// SIMATIC STEP 7 (V5.x) project Combined_DEH_Config
// station: P_ADR_BUS
// station: Hardware
// station: SIMATIC 400(ATC-RSM)
// station: SIMATIC 400(OPC-OA)
// station: P_ADR_BUS
// station: Hardware
// program: S7 Program
// program: S7 Program(1)

SYMBOL_TABLE
"Constants_RSM"	DB 1	DB 1	// Sheet 2 (RSM)
"HISIGMTR-VALs"	DB 2	DB 2
"LOSIGMTR-VALs"	DB 3	DB 3
"AIN_VALs_VIB"	DB 4	FB 1	// DB for analog vibration inputs
"GAINBI-VALs"	DB 5	DB 5
"DELTAW-VALs"	DB 6	DB 6	// DELTAW contants
"HILOLMTV-VALs"	DB 7	DB 7
"HILOMTR-VALs"	DB 8	DB 8
"AVALGEN"	DB 9	DB 9	// Analog Value Generation
"DVALGEN"	DB 10	DB 10	// Digital Value Generation
"RUNAVG_VALs_369_370"	DB 11	FB 2	// RUNAVG_DB for blocks 369  and 370
"HISIGMTV-VALs"	DB 12	DB 12
"LOSIGMTV-VALs"	DB 13	DB 13
"XLIMIT_VALs"	DB 14	DB 14
"AIFCTGEN_Vals"	DB 15	DB 15
"MULTGB_VALs"	DB 16	DB 16
"SUM2W_VALs"	DB 17	DB 17
"RATEMTR_VALs"	DB 18	DB 18
"XSUM_VALs"	DB 19	DB 19
"XTRANSF_VALs"	DB 20	DB 20
"XHISEL_VALs"	DB 21	DB 21
"AIN_VALs_TEMP_100"	DB 22	FB 1
"DIVIDEGB_VALs"	DB 23	DB 23
"AIN_VALs_TEMP_286"	DB 24	FB 1
"POLY_VALs"	DB 25	DB 25
"SUM4W_VALs"	DB 26	DB 26
"SUM8W_VALs"	DB 27	DB 27
"AIN_VALs_TEMP_661"	DB 28	FB 1	// DB for analog temperature inputs
"AIN_VALs_PRESS_760"	DB 29	FB 1	// DB for pressure analog inputs
"RESETSUM_VALs"	DB 30	DB 30
"AIN_VALs_POS_25"	DB 31	FB 1
"XMULT_VALs"	DB 32	DB 32
"ATCTime_VALs"	DB 33	DB 33	// Time declaration for all the timers used
"DIGCNTNF_VALs"	DB 34	DB 34
"Constants_ATC"	DB 35	DB 35
"RUNAVG_VALs_235"	DB 36	FB 2
"AIN_VALs_POS_2"	DB 37	FB 1	// DB for analog position inputs
"RSMTime_VALs"	DB 38	DB 38
"TIMECHG_VALs"	DB 39	DB 39
"AIN"	FB 1	FB 1	// REAL conversion of analog input signals
"RUNAVG"	FB 2	FB 2	// Average of time based samples of input
"DRUMD16"	FB 3	FB 3	// Drum Controller with Sixteen Digital Outputs
"QC"	FC 1	FC 1	// QCHK1BAD
"Sheet 24 (ATC)"	FC 2	FC 2	// VIBRATION MONITOR
"TOD_Conversion"	FC 3	FC 3	// Supporting Block for Sheet 24 (ATC)
"Sheet 2 (RSM)"	FC 4	FC 4	// Initialization of constants in sheet 2 (RSM)
"TRANSF"	FC 5	FC 5	// Transfer between Two Analog Inputs
"AIFCTGEN"	FC 6	FC 6
"BIN_SEARCH"	FC 7	FC 7
"XHISEL"	FC 8	FC 8	// Selects the Greater of Two Gained and Biased Inputs
"QAVGN"	FC 10	FC 10	// Average up to Eight Analog Points
"HISIGMTR"	FC 11	FC 11	// High Signal Monitor with Reset Deadband and Fixed Limit
"LOSIGMTR"	FC 12	FC 12	// Low Signal Monitor with Reset Deadband and Fixed Limit
"GAINBI"	FC 14	FC 14	// Gain and Bias an Input
"DELTAW"	FC 15	FC 15	// Difference between Two Weighted Inputs
"HILOLMTV"	FC 16	FC 16	// High/Low Limiter, Variable Limits
"HILOMTR"	FC 18	FC 18	// High/Low Signal Monitor with Reset Deadband and Fixed Limits
"QTRANSN"	FC 19	FC 19	// Automatic transfer between analog inputs, select best quality
"DIVIDEGB"	FC 21	FC 21	// Divider with Gain and Bias
"POLY"	FC 22	FC 22	// Fifth Order Polynomial Equation
"QBLOCK"	FC 23	FC 23	// Output is equal to input and output quality is good.
"SUM8W"	FC 24	FC 24
"Sheet 3 (RSM)"	FC 25	FC 25	// FSST & TIMP & TSAT (Analog)
"Sheet 4 (RSM)"	FC 26	FC 26	// HP FILM & TICM & TMAX (Analog)
"Sheet 5 (RSM)"	FC 27	FC 27	// MWINC LOGIC (Digital)
"Sheet 7 (RSM)"	FC 28	FC 28	// HP INVALID LOGIC (Digital)
"RESETSUM"	FC 29	FC 29	// Summer with Reset
"Sheet 6 (RSM)"	FC 30	FC 30	// HP Stress Counters (Analog)
"HISIGMTV"	FC 31	FC 31	// High Signal Monitor, Reset Deadband and Variable Limits
"LOSIGMTV"	FC 32	FC 32	// Low Signal Monitor, Reset Deadband, Variable Limit
"HISEL10"	FC 33	FC 33	// High Signal Selector with 'TWO' Inputs
"XLIMIT"	FC 34	FC 34	// Limits a Gained and Biased Input
"LOSEL10"	FC 35	FC 35	// Low Signal Selector with 'TWO' Inputs
"Sheet 9 (RSM)"	FC 36	FC 36	// HP ROTSURF, T1-5 & TP1-4 (Analog)
"Sheet 8 (RSM)"	FC 37	FC 37	// HXFER & TWC (Analog)
"Sheet 10 (RSM)"	FC 38	FC 38	// HP TEMP T6-T15 (Analog)
"Sheet11 (RSM)"	FC 39	FC 39	// HP TEMP T16-T23 (Analog)
"MULTGB"	FC 40	FC 40	// Multiplier with Gain and Bias
"SUM2W"	FC 41	FC 41	// Sum of Two Weighted Inputs
"RATEMTR"	FC 42	FC 42	// Rate of Change Monitor, Reset Deadband, Fixed Rate Limit
"XSUM"	FC 43	FC 43	// Add Two Gained and Biased Inputs
"XTRANSF"	FC 44	FC 44	// Select a Gained and Biased Input Based on a Flag
"Sheet 12 (RSM)"	FC 45	FC 45	// HP TAVG (Analog)
"Sheet 13 (RSM)"	FC 46	FC 46	// HP EFFECTIVE TEMP DIFF. (Analog)
"Sheet 14 (RSM)"	FC 47	FC 47	// HP DRUM TIMERS (Analog)
"Sheet 15 (RSM)"	FC 48	FC 48	// HP TD1FT1-15 (Analog)
"Sheet 16 (RSM)"	FC 51	FC 51	// HP ANTIC. DIFF. (Analog)
"Sheet 17 (RSM)"	FC 53	FC 53	// % ROTOR STRESS LIMIT (Analog)
"XMULT"	FC 54	FC 54	// Multiples Two Gained and Biased Inputs
"Sheet 18 (RSM)"	FC 55	FC 55	// SMW INC/DEC (Analog)
"Sheet 19 (RSM)"	FC 57	FC 57	// TBP (Analog)
"Sheet 20 (RSM)"	FC 58	FC 58	// MWINCR (Analog)
"Sheet 21 (RSM)"	FC 59	FC 59	// ATC RATE & LOAD RESERVE (Analog)
"SUM4W"	FC 60	FC 60
"Sheet 22 (RSM)"	FC 61	FC 61	// REQ. STM CHEST METAL TEMP (Analog)
"Sheet 23 (RSM)"	FC 62	FC 62	// HP ROTOR STRESS LIMIT (Digital)
"Sheet 24 (RSM)"	FC 63	FC 63	// ATC TARGET (Analog)
"Sheet 25 (RSM)"	FC 64	FC 64	// TRANSFER DELAY (Digital)
"Sheet 26 (RSM)"	FC 65	FC 65	// LADDERS 35, 128, RESONANCE RANGE LOGIC (Digital)
"Sheet 28 (RSM)"	FC 66	FC 66	// LADDERS 22, 500, 600, DIGITAL POINTERS TMAX & TWC LOGIC (Digital)
"Sheet 29 (RSM)"	FC 67	FC 67	// LADDERS 29, 31, 500, FIRST STAGE STM > 75 *C (Digital)
"Sheet 27 (RSM)"	FC 68	FC 68	// LADDERS 43, 129, RTSHOLD (Digital)
"Sheet 30 (RSM)"	FC 69	FC 69	// LADDER 126, SYNC LOGIC & OVERRIDE (Digital)
"Sheet 31 (RSM)"	FC 70	FC 70	// LADDER 33, ANTIC HP STRESS > LIMIT (Digital)
"Sheet 32 (RSM)"	FC 71	FC 71	// LADDERS 37, 125, 130, SYNC LOGIC & OVERRIDE (Digital)
"Sheet 33 (RSM)"	FC 72	FC 72	// LADDER 124, 127, SYNC LOGIC & TVGVINIT (Digital)
"Sheet 34 (RSM)"	FC 73	FC 73	// LADDERS 122, 123, 135, SET SPEED PLATEAU (Digital)
"Sheet 35 (RSM)"	FC 74	FC 74	// LADDER 120, 121, P15 ALARMS ESTIMATE ROLL TIME LOGIC & ATC VPL (Digital)
"Sheet 36 (RSM)"	FC 75	FC 75	// LADDER 41, 119, P15 ALARMS (Digital)
"Sheet 37 (RSM)"	FC 76	FC 76	// GENERATOR AND EXCITOR TEMPERATURES (Analog)
"Sheet 2 (ATC)"	FC 77	FC 77	// LADDER 500, SENSOR FAIL (Digital)
"Sheet 3 (ATC)"	FC 78	FC 78	// SENSOR FAIL (Digital)
"DIGCNTNF"	FC 79	FC 79	// Digital Counter with Flag
"Sheet 4 (ATC)"	FC 81	FC 81	// LADDERS 1, 3 (Digital)
"Sheet 5 (ATC)"	FC 82	FC 82	// LADDERS 3, 5, 9, 600, P00M01-M11 (Digital)
"Sheet 6 (ATC)"	FC 83	FC 83	// LADDERS 7, 9, 13, ATC PERMISSIVE (Digital)
"Sheet 7 (ATC)"	FC 84	FC 84	// LADDER 81. LOOPS 27, 33. WATER COOLED GENERATOR (Analog)
"Sheet 8 (ATC)"	FC 85	FC 85	// LADDERS 91, 108, 133, GENERATOR ANNUNCIATOR (Digital)
"Sheet 9 (ATC)"	FC 86	FC 86	// LADDERS 81,83,85,87,109,130. LOOPS 28-30. EXMON & COOLGSHI & P09MXX  (Digital)
"Sheet 10 (ATC)"	FC 87	FC 87	// LADDERS 31, 34, 36, GENERATOR CALCULATIONS (Analog)
"Sheet 11 (ATC)"	FC 88	FC 88	// LADDERS 15, 17, 18. LOOPS 2, 3. STEAM CHEST - OIL COOLER MONITOR (Analog)
"2xHISIGMTV, QC"	FC 89	FC 89	// Supporting block for sheet 12, 24 (ATC)
"Sheet 12 (ATC)"	FC 91	FC 91	// BEARING METAL TEMPERATURES (Analog)
"Sheet 13 (ATC)"	FC 92	FC 92	// BEARING METAL, OIL COOLER - P08MXX (Digital)
"Sheet 14 (ATC)"	FC 93	FC 93	// BEARING METAL - P08M05, 8 (Digital)
"Sheet 15 (ATC)"	FC 94	FC 94	// ROTOR POSITION, DIFF EXPANSION (Analog)
"Sheet 16 (ATC)"	FC 95	FC 95	// ROTOR POSITION DIFFERENTIAL EXPANSION P11MXX (Digital)
"Sheet 17 (ATC)"	FC 96	FC 96	// LOOPS 39, 40, 41. CONDENSOR PRESS LP EXH HOOD (Analog)
"Sheet 18 (ATC)"	FC 97	FC 97	// LADDERS 89, 90, 189, 190. GLAND, EXH, VAC - P10MXX (Digital)
"Sheet 19 (ATC)"	FC 98	FC 98	// BRG TEMPERATURE HIGH & VBINC (Digital)
"Sheet 20 (ATC)"	FC 99	FC 99	// VIBRATION LIMIT (Analog)
"Sheet 21 (ATC)"	FC 100	FC 100	// LADDERS 302,304,306,400. VIBRATION ALARM AND TRIP (Digital)
"Sheet 22 (ATC)"	FC 101	FC 101	// LADDERS 32, 33, 41. VIBRATION RUNUP / RUNDOWN LOGIC (Digital)
"Sheet 23 (ATC)"	FC 102	FC 102	// LADDER 39. VIBRATION RUNDOWN / RUNBACK LOGIC (Digital)
"3xHISIGMTV, 1xLOSIGMTV"	FC 103	FC 103
"3xLOSIGMTV, 1xHISIGMTV"	FC 104	FC 104
"SCALE"	FC 105	FC 105	// Scaling Values
"Sheet 25 (ATC)"	FC 106	FC 106	// SPEED RESONANT RANGE MONITOR (Analog)
"Sheet 26 (ATC)"	FC 107	FC 107	// LADDERS 150, 420. VIBRATION SPEED REF LOGIC (Digital)
"Sheet 27 (ATC)"	FC 108	FC 108	// VIBRATION RUNBACK SPEED REF (Analog)
"Sheet 28 (ATC)"	FC 109	FC 109	// LADDERS 30, 43, 307, 308, 309. VIBRATION RUNUP/RUNTHRU LOGIC (Digital)
"Sheet 29 (ATC)"	FC 110	FC 110	// VIBRATION RUN THRU REF (Analog)
"Sheet 30 (ATC)"	FC 111	FC 111	// VIBRATION SPEED REF (Analog)
"Sheet 31 (ATC)"	FC 112	FC 112	// LOOPS 18, 19. WATER DETECTION (Analog)
"Sheet 32 (ATC)"	FC 113	FC 113	// LADDERS 49, 51, 53. DRAIN VALVE LOGIC (Digital)
"DT_TOD"	FC 115	FC 115	// DT to TOD
"SUBB24"	FC 116	FC 116	// Supporting block for sheet 24 (ATC)
"TIMECHG"	FC 117	FC 117	// Check Real-Time Clock, Set Flags
"Sheet 33 (ATC)"	FC 118	FC 118	// LOOPS 4, 5 (Analog)
"Sheet 34 (ATC)"	FC 119	FC 119	// LADDERS 19, 21, 23, 25, 27. TURNING GEAR - P03MXX (Digital)
"Sheet 35 (ATC)"	FC 120	FC 120	// LOOPS 6, 60. THRUST BEARING, ROTOR ECCEN. (Analog)
"Sheet 36 (ATC)"	FC 121	FC 121	// LADDERS 27, 600. ATC PLATEAU FLAGS (Digital)
"Sheet 37 (ATC)"	FC 122	FC 122	// OVERRIDE LOGIC (Analog)
"Sheet 38 (ATC)"	FC 123	FC 123	// OVERRIDE LOGIC (Digital)
"Sheet 39 (ATC)"	FC 124	FC 124	// OVERRIDE LOGIC (Digital)
"Sheet 40 (ATC)"	FC 125	FC 125	// LADDERS 200, 201, 203, 220. REQUEST TRIP P07MXX (Digital)
"Sheet 41 (ATC)"	FC 126	FC 126	// LADDERS 201, 202, 203. HOLD 1 & 2 - P07M13 (Digital)
"Sheet 42 (ATC)"	FC 127	FC 127	// LADDERS 110, 111, 112, 113. OVERRIDE & P07M12 (Digital)
"Sheet 43 (ATC)"	FC 128	FC 128	// LADDERS 11, 113, 114. HOLD LOAD & P07M09 - 14 (Digital)
"Sheet 44 (ATC)"	FC 129	FC 129	// LADDERS 115, 116. HOLD WS & P07M02 - 04 (Digital)
"Sheet 45 (ATC)"	FC 130	FC 130	// LADDERS 117, 118. LOAD RATE INC/DEC P07M05 - 08 (Digital)
"Sheet 47 (ATC)"	FC 131	FC 131	// LADDERS 118, 192. P00M00A-G (Digital)
"Sheet 46 (ATC)"	FC 132	FC 132	// LOOPS 63, 65. LOAD RATE (Analog)
"Sheet 48_49 (ATC)"	FC 133	FC 133	// Initialization of ATC constants from AVALGEN DB
"ASSAP"	I 0.0	BOOL	//  (ATC) - (FieldIO4-M1)
"BOPL"	I 0.1	BOOL	//  (ATC) - (FieldIO4-M1)
"BVAP"	I 0.2	BOOL	//  (ATC) - (FieldIO4-M1)
"DVSAP"	I 0.3	BOOL	//  (ATC) - (FieldIO4-M1)
"EHFPL"	I 0.4	BOOL	//  (ATC) - (FieldIO4-M1)
"EHSO"	I 0.5	BOOL	//  (ATC) - (FieldIO4-M1)
"GDOGF"	I 0.6	BOOL	//  (ATC) - (FieldIO4-M1)
"GVRNLV"	I 0.7	BOOL	//  (ATC) - (FieldIO4-M1)
"HPDVC"	I 1.0	BOOL	//  (ATC) - (FieldIO4-M1)
"HPDVO"	I 1.1	BOOL	//  (ATC) - (FieldIO4-M1)
"MBCSU"	I 1.2	BOOL	//  (ATC) - (FieldIO4-M1)
"MELIT"	I 1.3	BOOL	//  (ATC) - (FieldIO4-M1)
"MVHPIT"	I 1.4	BOOL	//  (ATC) - (FieldIO4-M1)
"OEPIT"	I 1.5	BOOL	//  (ATC) - (FieldIO4-M1)
"RSBC"	I 1.6	BOOL	//  (ATC) - (FieldIO4-M1)
"RSBSU"	I 1.7	BOOL	//  (ATC) - (FieldIO4-M1)
"TGE"	I 2.0	BOOL	//  (ATC) - (FieldIO5-M1)
"VRO"	I 2.1	BOOL	//  (ATC) - (FieldIO5-M1)
"VROUS"	I 2.2	BOOL	//  (ATC) - (FieldIO5-M1)
"VRSOTP"	I 2.3	BOOL	//  (ATC) - (FieldIO5-M1)
"CAB4T1_W"	IW 512	WORD	//  (RSM) - (FieldIO4-M3)
"CNDP1_W"	IW 514	WORD	//  (RSM) - (FieldIO4-M3)
"FSST1_W"	IW 516	WORD	//  (RSM) - (FieldIO4-M3)
"B1T1_W"	IW 518	WORD	//  (ATC) - (FieldIO4-M3)
"B2T1_W"	IW 520	WORD	//  (ATC) - (FieldIO4-M3)
"B3T1_W"	IW 522	WORD	//  (ATC) - (FieldIO4-M3)
"B4T1_W"	IW 524	WORD	//  (ATC) - (FieldIO4-M3)
"B5T1_W"	IW 526	WORD	//  (ATC) - (FieldIO4-M3)
"B6T1_W"	IW 528	WORD	//  (ATC) - (FieldIO4-M4)
"RP1_W"	IW 530	WORD	//  (ATC) - (FieldIO4-M4)
"TBFCT1_W"	IW 532	WORD	//  (ATC) - (FieldIO4-M4)
"TBFLT1_W"	IW 534	WORD	//  (ATC) - (FieldIO4-M4)
"TBRCT1_W"	IW 536	WORD	//  (ATC) - (FieldIO4-M4)
"TBRLT1_W"	IW 538	WORD	//  (ATC) - (FieldIO4-M4)
"VB9_W"	IW 540	WORD	//  (ATC) - (FieldIO4-M4)
"FSMT1_W"	IW 542	WORD	//  (RSM) - (FieldIO4-M4)
"B7T_W"	IW 544	WORD	//  (ATC) - (FieldIO4-M5)
"B8T_W"	IW 546	WORD	//  (ATC) - (FieldIO4-M5)
"B9T_W"	IW 548	WORD	//  (ATC) - (FieldIO4-M5)
"B10T_W"	IW 550	WORD	//  (ATC) - (FieldIO4-M5)
"CAB5T1_W"	IW 552	WORD	//  (ATC) - (FieldIO4-M5)
"CAB5T2_W"	IW 554	WORD	//  (ATC) - (FieldIO4-M5)
"CASEXP_W"	IW 556	WORD	//  (ATC) - (FieldIO4-M5)
"DEGEN_W"	IW 558	WORD	//  (ATC) - (FieldIO4-M5)
"VB1_W"	IW 560	WORD	//  (ATC) - (FieldIO4-M6)
"VB2_W"	IW 562	WORD	//  (ATC) - (FieldIO4-M6)
"VB3_W"	IW 564	WORD	//  (ATC) - (FieldIO4-M6)
"VB4_W"	IW 566	WORD	//  (ATC) - (FieldIO4-M6)
"VB5_W"	IW 568	WORD	//  (ATC) - (FieldIO4-M6)
"VB6_W"	IW 570	WORD	//  (ATC) - (FieldIO4-M6)
"VB7_W"	IW 572	WORD	//  (ATC) - (FieldIO4-M6)
"VB8_W"	IW 574	WORD	//  (ATC) - (FieldIO4-M6)
"CAB4T2_W"	IW 576	WORD	//  (RSM) - (FieldIO5-M3)
"CNDP2_W"	IW 578	WORD	//  (RSM) - (FieldIO5-M3)
"FSST2_W"	IW 580	WORD	//  (RSM) - (FieldIO5-M3)
"B1T2_W"	IW 582	WORD	//  (ATC) - (FieldIO5-M3)
"B2T2_W"	IW 584	WORD	//  (ATC) - (FieldIO5-M3)
"B3T2_W"	IW 586	WORD	//  (ATC) - (FieldIO5-M3)
"B4T2_W"	IW 588	WORD	//  (ATC) - (FieldIO5-M3)
"B5T2_W"	IW 590	WORD	//  (ATC) - (FieldIO5-M3)
"B6T2_W"	IW 592	WORD	//  (ATC) - (FieldIO5-M4)
"RP2_W"	IW 594	WORD	//  (ATC) - (FieldIO5-M4)
"TBFCT2_W"	IW 596	WORD	//  (ATC) - (FieldIO5-M4)
"TBFLT2_W"	IW 598	WORD	//  (ATC) - (FieldIO5-M4)
"TBRCT2_W"	IW 600	WORD	//  (ATC) - (FieldIO5-M4)
"TBRLT2_W"	IW 602	WORD	//  (ATC) - (FieldIO5-M4)
"VB10_W"	IW 604	WORD	//  (ATC) - (FieldIO5-M4)
"LPGST_W"	IW 606	WORD	//  (RSM) - (FieldIO5-M4)
"EHFLT_W"	IW 608	WORD	//  (ATC) - (FieldIO5-M5)
"HPBMIDT_W"	IW 610	WORD	//  (ATC) - (FieldIO5-M5)
"HPCMIDT_W"	IW 612	WORD	//  (ATC) - (FieldIO5-M5)
"LP1GNT_W"	IW 614	WORD	//  (ATC) - (FieldIO5-M5)
"LP1GVT_W"	IW 616	WORD	//  (ATC) - (FieldIO5-M5)
"LP2GNT_W"	IW 618	WORD	//  (ATC) - (FieldIO5-M5)
"LP2GVT_W"	IW 620	WORD	//  (ATC) - (FieldIO5-M5)
"ROTECC_W"	IW 622	WORD	//  (ATC) - (FieldIO5-M5)
"OCIT_W"	IW 624	WORD	//  (RSM) - (FieldIO5-M6)
"OCOT_W"	IW 626	WORD	//  (RSM) - (FieldIO5-M6)
"TIMPRAT"	M 0.1	BOOL	// Sheet 3 (RSM)
"Z061"	M 0.2	BOOL	// Sheet 3 (RSM)
"Z060"	M 0.3	BOOL	// Sheet 3 (RSM)
"Z115"	M 0.4	BOOL	// Sheet 28 (RSM)
"SELC06"	M 0.5	BOOL	// Sheet 28 (RSM)
"X66D"	M 0.6	BOOL	// Sheet 4 (RSM)
"X67D"	M 0.7	BOOL	// Sheet 4 (RSM)
"X08A"	M 1.0	BOOL	// Sheet 4 (RSM)
"Z121"	M 1.1	BOOL	// Sheet 4 (RSM)
"Z133"	M 1.2	BOOL	// Sheet 4 (RSM)
"Z745"	M 1.3	BOOL	// Sheet 5 (RSM)
"Z747"	M 1.4	BOOL	// Sheet 5 (RSM)
"X08F"	M 1.5	BOOL	// Sheet 5 (RSM)
"X08E"	M 1.6	BOOL	// Sheet 5 (RSM)
"Z135"	M 1.7	BOOL	// Sheet 5 (RSM)
"Z393"	M 2.0	BOOL	// Sheet 19 (RSM)
"Z395"	M 2.1	BOOL	// Sheet 19 (RSM)
"Z398"	M 2.2	BOOL	// Sheet 19 (RSM)
"Z600"	M 2.3	BOOL	// Sheet 21 (RSM)
"BR"	M 2.4	BOOL	// Sheet 12 (OPC)
"Z599"	M 2.5	BOOL	// Sheet 21 (RSM)
"BR4"	M 2.6	BOOL	// Sheet 28 (RSM)
"F5MNLCTL"	M 2.7	BOOL	// Sheet 8 (RSM)
"Z272"	M 3.0	BOOL	// Sheet 6 (RSM)
"Z274"	M 3.1	BOOL	// Sheet 6 (RSM)
"WSFAIL"	M 3.2	BOOL	// Sheet 5 (OPC)
"HPINV"	M 3.3	BOOL	// Sheet 6 (RSM)
"RTRSWSFL"	M 3.4	BOOL	// Sheet 6 (RSM)
"Z268"	M 3.5	BOOL	// Sheet 7 (RSM)
"Z269"	M 3.6	BOOL	// Sheet 7 (RSM)
"Z123"	M 3.7	BOOL	// Sheet 7 (RSM)
"Z124"	M 4.0	BOOL	// Sheet 7 (RSM)
"P01M05"	M 4.1	BOOL	// Sheet 7 (RSM)
"Z131"	M 4.2	BOOL	// Sheet 7 (RSM)
"RESTART"	M 4.3	BOOL	// Sheet 7 (RSM)
"TIMPFAIL"	M 4.4	BOOL	// Sheet 7 (RSM)
"BRN4"	M 4.5	BOOL	// Sheet 28 (RSM)
"OUT_180"	M 4.6	BOOL	// Sheet 7 (RSM)
"X08D"	M 4.7	BOOL	// Sheet 6 (RSM)
"OUT_270"	M 5.0	BOOL	// Sheet 6 (RSM)
"T5SEC"	M 5.1	BOOL	// Sheet 6 (RSM)
"XFER"	M 5.2	BOOL	// Sheet 28 (RSM)
"OUT_221"	M 5.3	BOOL	// Sheet 8 (RSM)
"Z228"	M 5.4	BOOL	// Sheet 8 (RSM)
"X10G"	M 5.5	BOOL	// Sheet 11 (RSM)
"A275"	M 5.7	BOOL	// Sheet 14 (RSM)
"B275"	M 6.0	BOOL	// Sheet 14 (RSM)
"C275"	M 6.1	BOOL	// Sheet 14 (RSM)
"D275"	M 6.2	BOOL	// Sheet 14 (RSM)
"E275"	M 6.3	BOOL	// Sheet 14 (RSM)
"F275"	M 6.4	BOOL	// Sheet 14 (RSM)
"G275"	M 6.5	BOOL	// Sheet 14 (RSM)
"H275"	M 6.6	BOOL	// Sheet 14 (RSM)
"I275"	M 6.7	BOOL	// Sheet 14 (RSM)
"J275"	M 7.0	BOOL	// Sheet 14 (RSM)
"K275"	M 7.1	BOOL	// Sheet 14 (RSM)
"L275"	M 7.2	BOOL	// Sheet 14 (RSM)
"M275"	M 7.3	BOOL	// Sheet 14 (RSM)
"N275"	M 7.4	BOOL	// Sheet 14 (RSM)
"O275"	M 7.5	BOOL	// Sheet 14 (RSM)
"X11L"	M 7.6	BOOL	// Sheet 17 (RSM)
"X73K"	M 7.7	BOOL	// Sheet 17 (RSM)
"X11P"	M 8.0	BOOL	// Sheet 17 (RSM)
"X11T"	M 8.1	BOOL	// Sheet 17 (RSM)
"X11N"	M 8.2	BOOL	// Sheet 17 (RSM)
"X11R"	M 8.3	BOOL	// Sheet 17 (RSM)
"X11V"	M 8.4	BOOL	// Sheet 17 (RSM)
"X09L"	M 8.5	BOOL	// Sheet 17 (RSM)
"X09K"	M 8.6	BOOL	// Sheet 17 (RSM)
"X67A"	M 8.7	BOOL	// Sheet 17 (RSM)
"X14M"	M 9.0	BOOL	// Sheet 18 (RSM)
"X14Q"	M 9.1	BOOL	// Sheet 18 (RSM)
"P04CALC"	M 9.2	BOOL	// Sheet 21 (RSM)
"Z324"	M 9.3	BOOL	// Sheet 21 (RSM)
"Z325"	M 9.4	BOOL	// Sheet 21 (RSM)
"OUT_X73M"	M 9.5	BOOL	// Sheet 21 (RSM)
"NX1"	M 9.6	BOOL	// Sheet 22 (ATC)
"P07M03"	M 9.7	BOOL	// Sheet 44 (ATC)
"ATC4"	M 10.0	BOOL	// Sheet 28 (RSM)
"RUNBACK"	M 10.1	BOOL	// Sheet 23 (ATC)
"HOLD1"	M 10.2	BOOL	// Sheet 41 (ATC)
"HOLD2"	M 10.3	BOOL	// Sheet 41 (ATC)
"HILDPB"	M 10.4	BOOL	// Sheet 23 (RSM)
"NORLDPB"	M 10.5	BOOL	// Sheet 23 (RSM)
"LDEQDMD"	M 10.6	BOOL	// Sheet 5 (ATC)
"RBACK"	M 10.7	BOOL	// Sheet 23 (RSM)
"P01M02"	M 11.0	BOOL	// Sheet 23 (RSM)
"HILDRAT"	M 11.1	BOOL	// Sheet 23 (RSM)
"HLD1"	M 11.2	BOOL	// Sheet 27 (RSM)
"RES1"	M 11.3	BOOL	// Sheet 26 (RSM)
"RES2"	M 11.4	BOOL	// Sheet 26 (RSM)
"RES3"	M 11.5	BOOL	// Sheet 26 (RSM)
"RES4"	M 11.6	BOOL	// Sheet 26 (RSM)
"RES5"	M 11.7	BOOL	// Sheet 26 (RSM)
"EXC1"	M 12.0	BOOL	// Sheet 26 (RSM)
"P15M13"	M 12.1	BOOL	// Sheet 34 (RSM)
"DEHDMD1"	M 12.2	BOOL	// Sheet 35 (RSM)
"DEHDMD0"	M 12.3	BOOL	// Sheet 35 (RSM)
"AFLAG"	M 12.4	BOOL	// Sheet 25 (RSM)
"CRSBO4"	M 12.5	BOOL	// Sheet 25 (RSM)
"Z871"	M 12.6	BOOL	// Sheet 25 (RSM)
"HPPT2"	M 12.7	BOOL	// Sheet 31 (RSM)
"P04M03"	M 13.0	BOOL	// Sheet 31 (RSM)
"HPPT1"	M 13.1	BOOL	// Sheet 31 (RSM)
"HPPT3"	M 13.2	BOOL	// Sheet 31 (RSM)
"HOLDWS"	M 13.3	BOOL	// Sheet 44 (ATC)
"REQTRIP"	M 13.4	BOOL	// Sheet 40 (ATC)
"ASL4"	M 13.5	BOOL	// Sheet 28 (RSM)
"INRNG1"	M 13.6	BOOL	// Sheet 22 (ATC)
"INRNG2"	M 13.7	BOOL	// Sheet 22 (ATC)
"INRNG3"	M 14.0	BOOL	// Sheet 22 (ATC)
"INRNG4"	M 14.1	BOOL	// Sheet 22 (ATC)
"INEXC"	M 14.2	BOOL	// Sheet 22 (ATC)
"INRNG5"	M 14.3	BOOL	// Sheet 22 (ATC)
"HPRSHOLD"	M 14.4	BOOL	// Sheet 26 (RSM)
"HPRSIRAT"	M 14.5	BOOL	// Sheet 26 (RSM)
"HPSRATE"	M 14.6	BOOL	// Sheet 26 (RSM)
"P01M01"	M 14.7	BOOL	// Sheet 26 (RSM)
"TEMP_1"	M 15.0	BOOL	// Temporary variable for Sheet 26 (RSM)
"ASL"	M 15.1	BOOL	// Sheet 13 (OPC)
"ATC"	M 15.2	BOOL	// Sheet 12 (OA)
"BRX4"	M 15.3	BOOL	// Sheet 28 (RSM)
"RUNP04"	M 15.4	BOOL	// Sheet 29 (RSM)
"RUNTIMP"	M 15.5	BOOL	// Sheet 29 (RSM)
"TIMPHOLD"	M 15.6	BOOL	// Sheet 29 (RSM)
"P04M01"	M 15.7	BOOL	// Sheet 29 (RSM)
"HPRSRRAT"	M 16.0	BOOL	// Sheet 31 (RSM)
"HOLDLOAD"	M 16.1	BOOL	// Sheet 43 (ATC)
"BFLAG"	M 16.2	BOOL	// Sheet 33 (RSM)
"RTSHOLD"	M 16.3	BOOL	// Sheet 27 (RSM)
"RSREDRAT"	M 16.4	BOOL	// Sheet 27 (RSM)
"STHLDWS"	M 16.5	BOOL	// Sheet 27 (RSM)
"HLDONEWS"	M 16.6	BOOL	// Sheet 27 (RSM)
"P15M02"	M 16.7	BOOL	// Sheet 27 (RSM)
"ABFLAGT"	M 17.0	BOOL	// Sheet 27 (RSM)
"P15M25"	M 17.1	BOOL	// Sheet 32 (RSM)
"P15M06"	M 17.2	BOOL	// Sheet 36 (RSM)
"OVRDB"	M 17.3	BOOL	// PB 989, Sheet 30 (RSM)
"SYNCPROG"	M 17.4	BOOL	// Sheet 34 (RSM)
"CFLAG"	M 17.5	BOOL	// Sheet 33 (RSM)
"VBALM"	M 17.6	BOOL	// Sheet 21 (ATC)
"TEMP_2"	M 17.7	BOOL	// Temporary variable for Sheet 30 (RSM)
"TEMP_3"	M 18.0	BOOL	// Temporary variable for Sheet 30 (RSM)
"TEMP_4"	M 18.1	BOOL	// Temporary variable for Sheet 30 (RSM)
"TEMP_5"	M 18.2	BOOL	// Temporary variable for Sheet 30 (RSM)
"TEMP_6"	M 18.3	BOOL	// Temporary variable for Sheet 30 (RSM)
"OVRDPERM"	M 18.4	BOOL	// Sheet 30 (RSM)
"OVRDPB"	M 18.5	BOOL	// Sheet 30 (RSM)
"P15M21"	M 18.6	BOOL	// Sheet 30 (RSM)
"P15M22"	M 18.7	BOOL	// Sheet 30 (RSM)
"P15M23"	M 19.0	BOOL	// Sheet 30 (RSM)
"P15M24"	M 19.1	BOOL	// Sheet 30 (RSM)
"CNODE"	M 19.2	BOOL	// Sheet 30 (RSM)
"TEMP_7"	M 19.3	BOOL	// Temporary variable for Sheet 31 (RSM)
"TEMP_8"	M 19.4	BOOL	// Temporary variable for Sheet 31 (RSM)
"TEMP_9"	M 19.5	BOOL	// Temporary variable for Sheet 31 (RSM)
"EXCMON"	M 19.6	BOOL	// Sheet 9 (ATC)
"X65K"	M 19.7	BOOL	// Sheet 46 (ATC)
"TEMP_10"	M 20.0	BOOL	// Temporary variable for Sheet 32 (RSM)
"P15M19"	M 20.2	BOOL	// Sheet 32 (RSM)
"P15M20"	M 20.3	BOOL	// Sheet 32 (RSM)
"FSSTLTSF"	M 20.4	BOOL	// Sheet 32 (RSM)
"P15M10"	M 20.5	BOOL	// Sheet 32 (RSM)
"P15M14"	M 20.7	BOOL	// Sheet 33 (RSM)
"TEMP_11"	M 21.0	BOOL	// Sheet 33 (RSM)
"TEMP_12"	M 21.1	BOOL	// Sheet 33 (RSM)
"P15M15"	M 21.2	BOOL	// Sheet 33 (RSM)
"P15M16"	M 21.3	BOOL	// Sheet 33 (RSM)
"P15M17"	M 21.4	BOOL	// Sheet 33 (RSM)
"ATCASPB"	M 21.5	BOOL	// Sheet 33 (RSM)
"P15M18"	M 21.6	BOOL	// Sheet 33 (RSM)
"TEMP_13"	M 21.7	BOOL	// Sheet 33 (RSM)
"TRCOM"	M 22.0	BOOL	// Sheet 24 (OA)
"P15M07T"	M 22.1	BOOL	// Sheet 36 (RSM)
"P15M08"	M 22.2	BOOL	// Sheet 36 (RSM)
"P15M07"	M 22.3	BOOL	// Sheet 35 (RSM)
"ESTROTIM"	M 22.4	BOOL	// Sheet 35 (RSM)
"ATSVPLPB"	M 22.5	BOOL	// Sheet 35 (RSM)
"P15M04"	M 22.6	BOOL	// Sheet 35 (RSM)
"ROTGNP"	M 22.7	BOOL	// Sheet 34 (ATC)
"ROTROTG"	M 23.0	BOOL	// Sheet 34 (ATC)
"SAMERATE"	M 23.1	BOOL	// Sheet 36 (RSM)
"RSINCRAT"	M 23.2	BOOL	// Sheet 36 (RSM)
"P15M01"	M 23.3	BOOL	// Sheet 36 (RSM)
"P15M03"	M 23.4	BOOL	// Sheet 36 (RSM)
"TEMP_14"	M 23.5	BOOL	// Temporary variable for Sheet 36 (RSM)
"TEMP_15"	M 23.6	BOOL	// Temporary variable for Sheet 36 (RSM)
"P15M05"	M 23.7	BOOL	// Sheet 36 (RSM)
"MWFAIL"	M 24.0	BOOL	// Sheet 3 (OPC)
"ATC5"	M 24.1	BOOL	// Sheet 2 (ATC)
"ATCN"	M 24.2	BOOL	// Sheet 2 (ATC)
"ATC5HOLD"	M 24.3	BOOL	// Sheet 2 (ATC)
"ASL5"	M 24.4	BOOL	// Sheet 2 (ATC)
"BR5"	M 24.5	BOOL	// Sheet 2 (ATC)
"GENFAIL"	M 24.6	BOOL	// Sheet 2 (ATC)
"Z001"	M 24.7	BOOL	// Sheet 15 (ATC)
"Z025"	M 25.0	BOOL	// Sheet 24 (ATC)
"Z026"	M 25.1	BOOL	// Sheet 24 (ATC)
"Z027"	M 25.2	BOOL	// Sheet 24 (ATC)
"Z028"	M 25.3	BOOL	// Sheet 24 (ATC)
"Z029"	M 25.4	BOOL	// Sheet 24 (ATC)
"Z030"	M 25.5	BOOL	// Sheet 24 (ATC)
"Z033"	M 25.6	BOOL	// Sheet 24 (ATC)
"Z034"	M 25.7	BOOL	// Sheet 24 (ATC)
"Z035"	M 26.0	BOOL	// Sheet 24 (ATC)
"Z019"	M 26.1	BOOL	// Sheet 24 (ATC)
"APVBTP1"	M 26.2	BOOL	// Sheet 24 (ATC)
"APVBTP2"	M 26.3	BOOL	// Sheet 24 (ATC)
"APVBTP3"	M 26.4	BOOL	// Sheet 24 (ATC)
"APVBTP4"	M 26.5	BOOL	// Sheet 24 (ATC)
"APVBTP5"	M 26.6	BOOL	// Sheet 24 (ATC)
"APVBTP6"	M 26.7	BOOL	// Sheet 24 (ATC)
"APVBTP7"	M 27.0	BOOL	// Sheet 24 (ATC)
"APVBTP8"	M 27.1	BOOL	// Sheet 24 (ATC)
"APVBTP9"	M 27.2	BOOL	// Sheet 24 (ATC)
"DEFAIL"	M 27.3	BOOL	// Sheet 3 (ATC)
"VIBFAIL"	M 27.5	BOOL	// Sheet 3 (ATC)
"ANTVBTP"	M 27.6	BOOL	// Sheet 3 (ATC)
"P05M05"	M 27.7	BOOL	// Sheet 3 (ATC)
"APVBTP10"	M 28.0	BOOL	// Sheet 3 (ATC)
"RP1FAIL"	M 28.1	BOOL	// Sheet 15 (ATC)
"RP2FAIL"	M 28.2	BOOL	// Sheet 15 (ATC)
"VSFL1"	M 28.3	BOOL	// Sheet 4 (ATC)
"VSFAIL"	M 28.4	BOOL	// Sheet 4 (ATC)
"ADS"	M 28.5	BOOL	// Sheet 12 (OA)
"X60N"	M 28.6	BOOL	// Sheet 35 (ATC)
"P00M10"	M 28.7	BOOL	// Sheet 5 (ATC)
"P00M01"	M 29.0	BOOL	// Sheet 5 (ATC)
"P00M02"	M 29.1	BOOL	// Sheet 5 (ATC)
"DP007A"	M 29.2	BOOL	// Sheet 5 (ATC)
"P00M03"	M 29.3	BOOL	// Sheet 5 (ATC)
"DP50054"	M 29.4	BOOL	// Sheet 5 (ATC)
"P00M04"	M 29.5	BOOL	// Sheet 5 (ATC)
"P00M06"	M 29.6	BOOL	// Sheet 5 (ATC)
"BRX5"	M 29.7	BOOL	// Sheet 5 (ATC)
"TEMP1"	M 30.0	BOOL	// Temporary variable for Sheet 5 (ATC)
"P07M01"	M 30.1	BOOL	// Sheet 40 (ATC)
"ATCPERM"	M 30.2	BOOL	// Sheet 6 (ATC)
"SSPROA"	M 30.3	BOOL	// Sheet 6 (ATC)
"REJECT"	M 30.4	BOOL	// Sheet 6 (ATC)
"OUT_X30K"	M 30.5	BOOL	// Sheet 7 (ATC)
"OUT_X30L"	M 30.6	BOOL	// Sheet 7 (ATC)
"P10M01"	M 30.7	BOOL	// Sheet 8 (ATC)
"P10M02"	M 31.0	BOOL	// Sheet 8 (ATC)
"P09M22"	M 31.1	BOOL	// Sheet 9 (ATC)
"P09M23"	M 31.2	BOOL	// Sheet 9 (ATC)
"P09M24"	M 31.3	BOOL	// Sheet 9 (ATC)
"P09M26"	M 31.4	BOOL	// Sheet 9 (ATC)
"P09M25"	M 31.5	BOOL	// Sheet 9 (ATC)
"X75H"	M 31.6	BOOL	// Sheet 10 (ATC)
"X75I"	M 31.7	BOOL	// Sheet 10 (ATC)
"X75J"	M 32.0	BOOL	// Sheet 10 (ATC)
"X20A"	M 32.1	BOOL	// Sheet 11 (ATC)
"X20B"	M 32.2	BOOL	// Sheet 11 (ATC)
"X20C"	M 32.3	BOOL	// Sheet 11 (ATC)
"X20D"	M 32.4	BOOL	// Sheet 11 (ATC)
"Z840"	M 32.5	BOOL	// Sheet 11 (ATC)
"X20E"	M 32.6	BOOL	// Sheet 11 (ATC)
"Z813"	M 32.7	BOOL	// Sheet 12 (ATC)
"Z008"	M 33.0	BOOL	// Sheet 12 (ATC)
"Z043"	M 33.1	BOOL	// Sheet 12 (ATC)
"Z009"	M 33.2	BOOL	// Sheet 12 (ATC)
"Z045"	M 33.3	BOOL	// Sheet 12 (ATC)
"Z821"	M 33.4	BOOL	// Sheet 12 (ATC)
"Z012"	M 33.5	BOOL	// Sheet 12 (ATC)
"Z046"	M 33.6	BOOL	// Sheet 12 (ATC)
"Z814"	M 33.7	BOOL	// Sheet 12 (ATC)
"Z015"	M 34.0	BOOL	// Sheet 12 (ATC)
"Z047"	M 34.1	BOOL	// Sheet 12 (ATC)
"Z822"	M 34.2	BOOL	// Sheet 12 (ATC)
"Z016"	M 34.3	BOOL	// Sheet 12 (ATC)
"Z048"	M 34.4	BOOL	// Sheet 12 (ATC)
"Z815"	M 34.5	BOOL	// Sheet 12 (ATC)
"Z018"	M 34.6	BOOL	// Sheet 12 (ATC)
"Z049"	M 34.7	BOOL	// Sheet 12 (ATC)
"Z823"	M 35.0	BOOL	// Sheet 12 (ATC)
"Z112"	M 35.1	BOOL	// Sheet 12 (ATC)
"Z829"	M 35.2	BOOL	// Sheet 12 (ATC)
"Z113"	M 35.3	BOOL	// Sheet 12 (ATC)
"Z816"	M 35.4	BOOL	// Sheet 12 (ATC)
"Z031"	M 35.5	BOOL	// Sheet 12 (ATC)
"Z032"	M 35.6	BOOL	// Sheet 12 (ATC)
"Z075"	M 35.7	BOOL	// Sheet 12 (ATC)
"Z824"	M 36.0	BOOL	// Sheet 12 (ATC)
"Z038"	M 36.1	BOOL	// Sheet 12 (ATC)
"Z076"	M 36.2	BOOL	// Sheet 12 (ATC)
"Z817"	M 36.3	BOOL	// Sheet 12 (ATC)
"Z241"	M 36.4	BOOL	// Sheet 12 (ATC)
"Z077"	M 36.5	BOOL	// Sheet 12 (ATC)
"Z825"	M 36.6	BOOL	// Sheet 12 (ATC)
"Z041"	M 36.7	BOOL	// Sheet 12 (ATC)
"Z078"	M 37.0	BOOL	// Sheet 12 (ATC)
"Z818"	M 37.1	BOOL	// Sheet 12 (ATC)
"Z042"	M 37.2	BOOL	// Sheet 12 (ATC)
"Z079"	M 37.3	BOOL	// Sheet 12 (ATC)
"Z826"	M 37.4	BOOL	// Sheet 12 (ATC)
"ZAA"	M 37.5	BOOL	// Sheet 12 (ATC)
"ZBB"	M 37.6	BOOL	// Sheet 12 (ATC)
"ZCC"	M 37.7	BOOL	// Sheet 12 (ATC)
"Z114"	M 38.0	BOOL	// Sheet 12 (ATC)
"Z830"	M 38.1	BOOL	// Sheet 12 (ATC)
"ZA115"	M 38.2	BOOL	// Sheet 12 (ATC)
"Z116"	M 38.3	BOOL	// Sheet 12 (ATC)
"Z831"	M 38.4	BOOL	// Sheet 12 (ATC)
"Z117"	M 38.5	BOOL	// Sheet 12 (ATC)
"Z360"	M 38.6	BOOL	// Sheet 12 (ATC)
"Z361"	M 38.7	BOOL	// Sheet 12 (ATC)
"Z836"	M 39.0	BOOL	// Sheet 12 (ATC)
"ZXX"	M 39.1	BOOL	// Sheet 12 (ATC)
"ZYY"	M 39.2	BOOL	// Sheet 12 (ATC)
"ZZZ"	M 39.3	BOOL	// Sheet 12 (ATC)
"Z362"	M 39.4	BOOL	// Sheet 12 (ATC)
"Z363"	M 39.5	BOOL	// Sheet 12 (ATC)
"Z832"	M 39.6	BOOL	// Sheet 12 (ATC)
"Z364"	M 39.7	BOOL	// Sheet 12 (ATC)
"Z365"	M 40.0	BOOL	// Sheet 12 (ATC)
"Z833"	M 40.1	BOOL	// Sheet 12 (ATC)
"Z366"	M 40.2	BOOL	// Sheet 12 (ATC)
"Z367"	M 40.3	BOOL	// Sheet 12 (ATC)
"Z834"	M 40.4	BOOL	// Sheet 12 (ATC)
"Z369"	M 40.5	BOOL	// Sheet 12 (ATC)
"Z370"	M 40.6	BOOL	// Sheet 12 (ATC)
"Z835"	M 40.7	BOOL	// Sheet 12 (ATC)
"Z371"	M 41.0	BOOL	// Sheet 12 (ATC)
"Z372"	M 41.1	BOOL	// Sheet 12 (ATC)
"Z838"	M 41.2	BOOL	// Sheet 12 (ATC)
"ZUU"	M 41.3	BOOL	// Sheet 12 (ATC)
"ZVV2"	M 41.4	BOOL	// Sheet 12 (ATC)
"ZWW"	M 41.5	BOOL	// Sheet 12 (ATC)
"Z052"	M 41.6	BOOL	// Sheet 12 (ATC)
"P08M05"	M 41.7	BOOL	// Sheet 14 (ATC)
"P08M08"	M 42.0	BOOL	// Sheet 14 (ATC)
"P08M01"	M 42.1	BOOL	// Sheet 13 (ATC)
"P08M02"	M 42.2	BOOL	// Sheet 13 (ATC)
"BRERR"	M 42.3	BOOL	// Sheet 13 (ATC)
"P08M09"	M 42.4	BOOL	// Sheet 13 (ATC)
"P08M03"	M 42.5	BOOL	// Sheet 13 (ATC)
"BMTTRIP"	M 42.6	BOOL	// Sheet 13 (ATC)
"P08M04"	M 42.7	BOOL	// Sheet 13 (ATC)
"P08M06"	M 43.0	BOOL	// Sheet 13 (ATC)
"P08M07"	M 43.1	BOOL	// Sheet 13 (ATC)
"BMTH"	M 43.2	BOOL	// Sheet 13 (ATC)
"P08M10"	M 43.3	BOOL	// Sheet 13 (ATC)
"X20H"	M 43.4	BOOL	// Sheet 17 (ATC)
"COIL81"	M 43.5	BOOL	// Sheet 14 (ATC)
"COIL82"	M 43.6	BOOL	// Sheet 14 (ATC)
"COIL83"	M 43.7	BOOL	// Sheet 14 (ATC)
"COIL84"	M 44.0	BOOL	// Sheet 14 (ATC)
"Z095"	M 44.1	BOOL	// Sheet 15 (ATC)
"Z270"	M 44.2	BOOL	// Sheet 15 (ATC)
"Z096"	M 44.3	BOOL	// Sheet 15 (ATC)
"Z271"	M 44.4	BOOL	// Sheet 15 (ATC)
"Z098"	M 44.5	BOOL	// Sheet 15 (ATC)
"Z273"	M 44.6	BOOL	// Sheet 15 (ATC)
"Z097"	M 44.7	BOOL	// Sheet 15 (ATC)
"ZA272"	M 45.0	BOOL	// Sheet 15 (ATC)
"Z106"	M 45.2	BOOL	// Sheet 15 (ATC)
"Z108"	M 45.3	BOOL	// Sheet 15 (ATC)
"Z089"	M 45.4	BOOL	// Sheet 15 (ATC)
"Z102"	M 45.5	BOOL	// Sheet 15 (ATC)
"Z090"	M 45.6	BOOL	// Sheet 15 (ATC)
"Z103"	M 45.7	BOOL	// Sheet 15 (ATC)
"DEOFFN"	M 46.0	BOOL	// Sheet 16 (ATC)
"DET"	M 46.1	BOOL	// Sheet 16 (ATC)
"P11M01"	M 46.2	BOOL	// Sheet 16 (ATC)
"P11M02"	M 46.3	BOOL	// Sheet 16 (ATC)
"DEHOLD"	M 46.4	BOOL	// Sheet 16 (ATC)
"P11M05"	M 46.5	BOOL	// Sheet 16 (ATC)
"P11M06"	M 46.6	BOOL	// Sheet 16 (ATC)
"ANDEHOLD"	M 46.7	BOOL	// Sheet 16 (ATC)
"P11M09"	M 47.0	BOOL	// Sheet 16 (ATC)
"RPOFFN"	M 47.1	BOOL	// Sheet 16 (ATC)
"P11M10"	M 47.2	BOOL	// Sheet 16 (ATC)
"X41D"	M 47.3	BOOL	// Sheet 17 (ATC)
"CONDHI"	M 47.4	BOOL	// Sheet 17 (ATC)
"Z137"	M 47.5	BOOL	// Sheet 17 (ATC)
"Z856"	M 47.6	BOOL	// Sheet 17 (ATC)
"Y2"	M 47.7	BOOL	// Sheet 17 (ATC)
"Y1"	M 48.0	BOOL	// Sheet 17 (ATC)
"Z845"	M 48.1	BOOL	// Sheet 17 (ATC)
"Z847"	M 48.2	BOOL	// Sheet 17 (ATC)
"X41A"	M 48.3	BOOL	// Sheet 17 (ATC)
"X41B"	M 48.4	BOOL	// Sheet 17 (ATC)
"Z846"	M 48.5	BOOL	// Sheet 17 (ATC)
"Z848"	M 48.6	BOOL	// Sheet 17 (ATC)
"P10M03"	M 48.7	BOOL	// Sheet 18 (ATC)
"EXHERR"	M 49.0	BOOL	// Sheet 18 (ATC)
"P10M04"	M 49.1	BOOL	// Sheet 18 (ATC)
"P10M05"	M 49.2	BOOL	// Sheet 18 (ATC)
"P10M08"	M 49.3	BOOL	// Sheet 18 (ATC)
"P10M09"	M 49.4	BOOL	// Sheet 18 (ATC)
"P10M06"	M 49.5	BOOL	// Sheet 18 (ATC)
"VACOFLIM"	M 49.6	BOOL	// Sheet 18 (ATC)
"P10M10"	M 49.7	BOOL	// Sheet 18 (ATC)
"VB1INC"	M 50.0	BOOL	// Sheet 24 (ATC)
"VB2INC"	M 50.1	BOOL	// Sheet 24 (ATC)
"VB3INC"	M 50.2	BOOL	// Sheet 24 (ATC)
"VB4INC"	M 50.3	BOOL	// Sheet 24 (ATC)
"VB5INC"	M 50.4	BOOL	// Sheet 24 (ATC)
"VB6INC"	M 50.5	BOOL	// Sheet 24 (ATC)
"VB7INC"	M 50.6	BOOL	// Sheet 24 (ATC)
"VB8INC"	M 50.7	BOOL	// Sheet 24 (ATC)
"VB9INC"	M 51.0	BOOL	// Sheet 24 (ATC)
"VB10INC"	M 51.1	BOOL	// Sheet 24 (ATC)
"VBCNT"	M 51.2	BOOL	// Sheet 24 (ATC)
"VRSCNP"	M 51.3	BOOL	// Sheet 21 (ATC)
"VBINC"	M 51.4	BOOL	// Sheet 19 (ATC)
"VBALM1"	M 51.5	BOOL	// Sheet 24 (ATC)
"VBALM2"	M 51.6	BOOL	// Sheet 24 (ATC)
"VBALM3"	M 51.7	BOOL	// Sheet 24 (ATC)
"VBALM4"	M 52.0	BOOL	// Sheet 24 (ATC)
"VBALM5"	M 52.1	BOOL	// Sheet 24 (ATC)
"VBALM6"	M 52.2	BOOL	// Sheet 24 (ATC)
"VBALM7"	M 52.3	BOOL	// Sheet 24 (ATC)
"VBALM8"	M 52.4	BOOL	// Sheet 24 (ATC)
"VBALM9"	M 52.5	BOOL	// Sheet 24 (ATC)
"VBALM10"	M 52.6	BOOL	// Sheet 24 (ATC)
"RBOS"	M 52.7	BOOL	// Sheet 28 (ATC)
"GOEXC"	M 53.0	BOOL	// Sheet 26 (ATC)
"VBTRP1"	M 53.1	BOOL	// Sheet 24 (ATC)
"VBTRP2"	M 53.2	BOOL	// Sheet 24 (ATC)
"VBTRP3"	M 53.3	BOOL	// Sheet 24 (ATC)
"VBTRP4"	M 53.4	BOOL	// Sheet 24 (ATC)
"VBTRP5"	M 53.5	BOOL	// Sheet 24 (ATC)
"VBTRP6"	M 53.6	BOOL	// Sheet 24 (ATC)
"VBTRP7"	M 53.7	BOOL	// Sheet 24 (ATC)
"VBTRP8"	M 54.0	BOOL	// Sheet 24 (ATC)
"VBTRP9"	M 54.1	BOOL	// Sheet 24 (ATC)
"VBTRP10"	M 54.2	BOOL	// Sheet 24 (ATC)
"X22M"	M 54.3	BOOL	// Sheet 35 (ATC)
"VBREJ1"	M 54.4	BOOL	// Sheet 21 (ATC)
"RESET"	M 54.5	BOOL	// Sheet 21 (ATC)
"P05M03"	M 54.6	BOOL	// Sheet 21 (ATC)
"VBTRP"	M 54.7	BOOL	// Sheet 21 (ATC)
"P05M02"	M 55.0	BOOL	// Sheet 21 (ATC)
"P05M01"	M 55.1	BOOL	// Sheet 21 (ATC)
"RECCGT3"	M 55.2	BOOL	// Sheet 21 (ATC)
"VBALMA"	M 55.3	BOOL	// Sheet 21 (ATC)
"Z331"	M 55.4	BOOL	// Sheet 25 (ATC)
"Z337"	M 55.5	BOOL	// Sheet 25 (ATC)
"Z332"	M 55.6	BOOL	// Sheet 25 (ATC)
"Z338"	M 55.7	BOOL	// Sheet 25 (ATC)
"Z333"	M 56.0	BOOL	// Sheet 25 (ATC)
"Z339"	M 56.1	BOOL	// Sheet 25 (ATC)
"Z334"	M 56.2	BOOL	// Sheet 25 (ATC)
"Z340"	M 56.3	BOOL	// Sheet 25 (ATC)
"Z335"	M 56.4	BOOL	// Sheet 25 (ATC)
"Z341"	M 56.5	BOOL	// Sheet 25 (ATC)
"Z397"	M 56.6	BOOL	// Sheet 25 (ATC)
"ZA398"	M 56.7	BOOL	// Sheet 25 (ATC)
"RUNUP"	M 57.0	BOOL	// Sheet 28 (ATC)
"RUNTHRU"	M 57.1	BOOL	// Sheet 28 (ATC)
"RUNDOWN"	M 57.2	BOOL	// Sheet 23 (ATC)
"INRNG"	M 57.3	BOOL	// Sheet 22 (ATC)
"RDORIDE"	M 57.4	BOOL	// Sheet 22 (ATC)
"VBSTDY"	M 57.5	BOOL	// Sheet 22 (ATC)
"VBDEC"	M 57.6	BOOL	// Sheet 22 (ATC)
"NI"	M 57.7	BOOL	// Sheet 22 (ATC)
"P11SET"	M 58.0	BOOL	// Sheet 22 (ATC)
"P00M12"	M 58.1	BOOL	// Sheet 22 (ATC)
"P0M05"	M 58.2	BOOL	// Sheet 22 (ATC)
"HOLDSPD"	M 58.3	BOOL	// Sheet 22 (ATC)
"HSOTIME"	M 58.4	BOOL	// Sheet 22 (ATC)
"RBOK"	M 58.5	BOOL	// Sheet 26 (ATC)
"HLDWS"	M 58.6	BOOL	// Sheet 44 (ATC)
"RDEQASR"	M 58.7	BOOL	// Sheet 40 (ATC)
"TEMP2"	M 59.1	BOOL	// Temporary variable for Sheet 23 (ATC)
"Z714"	M 59.2	BOOL	// Sheet 23 (ATC)
"Z712"	M 59.3	BOOL	// Sheet 23 (ATC)
"TEMP3"	M 59.4	BOOL	// Temporary variable for Sheet 23 (ATC)
"P05M04"	M 59.5	BOOL	// Sheet 23 (ATC)
"TEMP4"	M 59.6	BOOL	// Temporary variable for Sheet 23 (ATC)
"Z415"	M 59.7	BOOL	// Sheet 25 (ATC)
"Z993"	M 60.0	BOOL	// Sheet 25 (ATC)
"Z864"	M 60.1	BOOL	// Sheet 25 (ATC)
"Z865"	M 60.2	BOOL	// Sheet 25 (ATC)
"Z867"	M 60.3	BOOL	// Sheet 25 (ATC)
"Z868"	M 60.4	BOOL	// Sheet 25 (ATC)
"Z870"	M 60.5	BOOL	// Sheet 25 (ATC)
"ZA871"	M 60.6	BOOL	// Sheet 25 (ATC)
"Z873"	M 60.7	BOOL	// Sheet 25 (ATC)
"Z874"	M 61.0	BOOL	// Sheet 25 (ATC)
"Z806"	M 61.1	BOOL	// Sheet 25 (ATC)
"Z807"	M 61.2	BOOL	// Sheet 25 (ATC)
"GTRTR1B"	M 61.3	BOOL	// Sheet 25 (ATC)
"LTRTR1T"	M 61.4	BOOL	// Sheet 25 (ATC)
"GTRTR2B"	M 61.5	BOOL	// Sheet 25 (ATC)
"LTRTR2T"	M 61.6	BOOL	// Sheet 25 (ATC)
"GTRTR3B"	M 61.7	BOOL	// Sheet 25 (ATC)
"LTRTR3T"	M 62.0	BOOL	// Sheet 25 (ATC)
"GTRTR4B"	M 62.1	BOOL	// Sheet 25 (ATC)
"LTRTR4T"	M 62.2	BOOL	// Sheet 25 (ATC)
"GTRTR5B"	M 62.3	BOOL	// Sheet 25 (ATC)
"LTRTR5T"	M 62.4	BOOL	// Sheet 25 (ATC)
"GTEXC1B"	M 62.5	BOOL	// Sheet 25 (ATC)
"LTEXC1T"	M 62.6	BOOL	// Sheet 25 (ATC)
"X01I"	M 62.7	BOOL	// Sheet 25 (ATC)
"Z349"	M 63.0	BOOL	// Sheet 25 (ATC)
"Z343"	M 63.1	BOOL	// Sheet 25 (ATC)
"Z350"	M 63.2	BOOL	// Sheet 25 (ATC)
"Z344"	M 63.3	BOOL	// Sheet 25 (ATC)
"Z351"	M 63.4	BOOL	// Sheet 25 (ATC)
"Z345"	M 63.5	BOOL	// Sheet 25 (ATC)
"Z352"	M 63.6	BOOL	// Sheet 25 (ATC)
"Z346"	M 63.7	BOOL	// Sheet 25 (ATC)
"Z353"	M 64.0	BOOL	// Sheet 25 (ATC)
"Z347"	M 64.1	BOOL	// Sheet 25 (ATC)
"RTHRUOK"	M 64.2	BOOL	// Sheet 26 (ATC)
"GO1"	M 64.3	BOOL	// Sheet 26 (ATC)
"GO2"	M 64.4	BOOL	// Sheet 26 (ATC)
"GO3"	M 64.5	BOOL	// Sheet 26 (ATC)
"GO4"	M 64.6	BOOL	// Sheet 26 (ATC)
"GO5"	M 64.7	BOOL	// Sheet 26 (ATC)
"PICK1"	M 65.0	BOOL	// Sheet 26 (ATC)
"PICK2"	M 65.1	BOOL	// Sheet 26 (ATC)
"PICK3"	M 65.2	BOOL	// Sheet 26 (ATC)
"PICK4"	M 65.3	BOOL	// Sheet 26 (ATC)
"PICK5"	M 65.4	BOOL	// Sheet 26 (ATC)
"PICKE"	M 65.5	BOOL	// Sheet 26 (ATC)
"PICKK1"	M 65.6	BOOL	// Sheet 26 (ATC)
"PICKK2"	M 65.7	BOOL	// Sheet 26 (ATC)
"PICKK3"	M 66.0	BOOL	// Sheet 26 (ATC)
"PICKK4"	M 66.1	BOOL	// Sheet 26 (ATC)
"PICKK5"	M 66.2	BOOL	// Sheet 26 (ATC)
"PICKKE"	M 66.3	BOOL	// Sheet 26 (ATC)
"RBSRIN1"	M 66.4	BOOL	// Sheet 26 (ATC)
"RBSRIN2"	M 66.5	BOOL	// Sheet 26 (ATC)
"RBSRIN3"	M 66.6	BOOL	// Sheet 26 (ATC)
"RBSRIN4"	M 66.7	BOOL	// Sheet 26 (ATC)
"RBSRIN5"	M 67.0	BOOL	// Sheet 26 (ATC)
"RBSRINEX"	M 67.1	BOOL	// Sheet 26 (ATC)
"Z696"	M 67.2	BOOL	// Sheet 30 (ATC)
"Z383"	M 67.3	BOOL	// Sheet 31 (ATC)
"Z379"	M 67.4	BOOL	// Sheet 31 (ATC)
"RBOSCL"	M 67.5	BOOL	// Sheet 28 (ATC)
"TEMP5"	M 67.6	BOOL	// Supporting varible for sheet 28 (ATC)
"GORUNUP"	M 67.7	BOOL	// Sheet 28 (ATC)
"RUNTHRUT"	M 68.0	BOOL	// Sheet 28 (ATC)
"H2OTRIP"	M 68.1	BOOL	// Sheet 28 (ATC)
"H2OHOLD"	M 68.2	BOOL	// Sheet 28 (ATC)
"P06M02"	M 68.3	BOOL	// Sheet 28 (ATC)
"RTORIDE"	M 68.4	BOOL	// Sheet 28 (ATC)
"P06M01"	M 68.5	BOOL	// Sheet 28 (ATC)
"OUT_695"	M 68.6	BOOL	// Sheet 30 (ATC)
"OUT_268"	M 68.7	BOOL	// Sheet 30 (ATC)
"Z919"	M 69.0	BOOL	// Sheet 28 (ATC)
"Z510"	M 69.1	BOOL	// Sheet 31 (ATC)
"Z505"	M 69.2	BOOL	// Sheet 31 (ATC)
"ZA119"	M 69.3	BOOL	// Sheet 31 (ATC)
"P06M09T"	M 69.4	BOOL	// Sheet 32 (ATC)
"P06M12T"	M 69.5	BOOL	// Sheet 32 (ATC)
"P06M06"	M 69.6	BOOL	// Sheet 32 (ATC)
"P06M05"	M 69.7	BOOL	// Sheet 32 (ATC)
"P06M03"	M 70.0	BOOL	// Sheet 32 (ATC)
"P06M04"	M 70.1	BOOL	// Sheet 32 (ATC)
"P06M07"	M 70.2	BOOL	// Sheet 32 (ATC)
"TEMP6"	M 70.3	BOOL	// Supporting varible for sheet 32 (ATC)
"X05G"	M 70.4	BOOL	// Sheet 33 (ATC)
"Z844"	M 70.5	BOOL	// Sheet 33 (ATC)
"P03M01"	M 70.6	BOOL	// Sheet 34 (ATC)
"ROTNP"	M 70.7	BOOL	// Sheet 34 (ATC)
"P03M02"	M 71.0	BOOL	// Sheet 34 (ATC)
"REQOV"	M 71.1	BOOL	// Sheet 34 (ATC)
"X60K"	M 71.2	BOOL	// Sheet 35 (ATC)
"ESPULS"	M 71.3	BOOL	// Sheet 36 (ATC)
"P03M03"	M 71.4	BOOL	// Sheet 36 (ATC)
"SYNCRNG"	M 71.5	BOOL	// Sheet 36 (ATC)
"SDNSYNC"	M 71.6	BOOL	// Sheet 36 (ATC)
"ES5"	M 71.7	BOOL
"ESX5"	M 72.0	BOOL	// Sheet 36 (ATC)
"OVRD1"	M 72.2	BOOL	// Sheet 37 (ATC)
"OVRD2"	M 72.3	BOOL	// Sheet 37 (ATC)
"OVRD3"	M 72.4	BOOL	// Sheet 37 (ATC)
"OVRD4"	M 72.5	BOOL	// Sheet 37 (ATC)
"OVRD5"	M 72.6	BOOL	// Sheet 38 (ATC)
"OVRD6"	M 72.7	BOOL	// Sheet 38 (ATC)
"OVRD7"	M 73.0	BOOL	// Sheet 38 (ATC)
"OVRD8"	M 73.1	BOOL	// Sheet 38 (ATC)
"OVRD9"	M 73.2	BOOL	// Sheet 38 (ATC)
"OVRD10"	M 73.3	BOOL	// Sheet 39 (ATC)
"OVRD11"	M 73.4	BOOL	// Sheet 39 (ATC)
"OVRD13"	M 73.5	BOOL	// Sheet 39 (ATC)
"P07M02"	M 73.6	BOOL	// Sheet 40 (ATC)
"X65I"	M 73.7	BOOL	// Sheet 46 (ATC)
"X65J"	M 74.0	BOOL	// Sheet 46 (ATC)
"P07M13"	M 74.1	BOOL	// Sheet 41 (ATC)
"REDOK"	M 74.2	BOOL	// Sheet 41 (ATC)
"INCOK"	M 74.3	BOOL	// Sheet 41 (ATC)
"OVRD20"	M 74.4	BOOL	// Sheet 42 (ATC)
"OVRD21"	M 74.5	BOOL	// Sheet 42 (ATC)
"OVRD22"	M 74.6	BOOL	// Sheet 42 (ATC)
"P07M12"	M 74.7	BOOL	// Sheet 42 (ATC)
"P07M14"	M 75.0	BOOL	// Sheet 43 (ATC)
"P07M10"	M 75.1	BOOL	// Sheet 43 (ATC)
"P07M09"	M 75.2	BOOL	// Sheet 43 (ATC)
"ATCHOLD"	M 75.3	BOOL	// Sheet 44 (ATC)
"P07M04"	M 75.4	BOOL	// Sheet 44 (ATC)
"Z861"	M 75.5	BOOL	// Sheet 44 (ATC)
"RATESEL"	M 75.6	BOOL	// Sheet 44 (ATC)
"RATETIME"	M 75.7	BOOL	// Sheet 45 (ATC)
"MOVERATE"	M 76.0	BOOL	// Sheet 45 (ATC)
"RATI8"	M 76.1	BOOL	// Sheet 45 (ATC)
"RATI4"	M 76.2	BOOL	// Sheet 45 (ATC)
"RATI3"	M 76.3	BOOL	// Sheet 45 (ATC)
"RATI2"	M 76.4	BOOL	// Sheet 45 (ATC)
"RATI1"	M 76.5	BOOL	// Sheet 45 (ATC)
"TEMP7"	M 76.6	BOOL	// Supporting varible for sheet 45 (ATC)
"P07M07"	M 76.7	BOOL	// Sheet 45 (ATC)
"P07M08"	M 77.0	BOOL	// Sheet 45 (ATC)
"P07M06"	M 77.1	BOOL	// Sheet 45 (ATC)
"P07M05"	M 77.2	BOOL	// Sheet 45 (ATC)
"TEMP8"	M 77.3	BOOL	// Supporting varible for sheet 47 (ATC)
"P00M00A"	M 77.4	BOOL	// Sheet 47 (ATC)
"P00M00B"	M 77.5	BOOL	// Sheet 47 (ATC)
"P00M00C"	M 77.6	BOOL	// Sheet 47 (ATC)
"P00M00D"	M 77.7	BOOL	// Sheet 47 (ATC)
"P00M00E"	M 78.0	BOOL	// Sheet 47 (ATC)
"P00M00G"	M 78.1	BOOL	// Sheet 47 (ATC)
"BRX5A"	M 78.2	BOOL	// Sheet 45 (ATC)
"TROOTHP"	M 78.3	BOOL	// Sheet 2 (RSM)
"VBHR"	M 78.4	BOOL	// Sheet 24 (ATC)
"VBSC"	M 78.5	BOOL	// Sheet 24 (ATC)
"FSST1"	MD 100	REAL	// Output of AIN block after FSST1 signal (Sheet 3)
"FSST2"	MD 104	REAL	// Output of AIN block after FSST2 signal (Sheet 3)
"FSST1E"	MD 108	REAL	// Sheet 3 (RSM)
"FSST2E"	MD 112	REAL	// Sheet 3 (RSM)
"OUT_369"	MD 116	REAL	// Sheet 3 (RSM)
"OUT_370"	MD 120	REAL	// Sheet 3 (RSM)
"OUT_371"	MD 124	REAL	// Sheet 3 (RSM)
"OUT_372"	MD 128	REAL	// Sheet 3 (RSM)
"OUT_374"	MD 132	REAL	// Sheet 3 (RSM)
"FSSTAVG"	MD 136	REAL	// Sheet 3 (RSM)
"FSSTLO"	MD 140	REAL	// Sheet 3 (RSM)
"TIMP1"	MD 144	REAL	// Sheet 3 (RSM)
"TIMP2"	MD 148	REAL	// Sheet 3 (RSM)
"Z119"	MD 152	REAL	// Sheet 3 (RSM)
"SAT"	MD 156	REAL	// Sheet 3 (RSM)
"TMAX"	MD 160	REAL	// Sheet 3 (RSM)
"TIMP"	MD 164	REAL	// Sheet 3 (RSM)
"OUT_793"	MD 168	REAL	// Sheet 3 (RSM)
"OUT_794"	MD 172	REAL	// Sheet 3 (RSM)
"TSAT"	MD 176	REAL	// Sheet 3 (RSM)
"Z104"	MD 180	REAL	// Sheet 4 (RSM)
"CNDP"	MD 184	REAL	// Sheet 4 (RSM)
"WS"	MD 188	REAL	// Sheet 4 (OPC)
"CONDPRES"	MD 192	REAL	// Sheet 3 (RSM)
"OUT_211"	MD 196	REAL	// Sheet 3 (RSM)
"OUT_212"	MD 200	REAL	// Sheet 3 (RSM)
"OUT_791"	MD 204	REAL	// Sheet 3 (RSM)
"PFS"	MD 208	REAL	// Sheet 3 (RSM)
"OUT_217"	MD 212	REAL	// Sheet 3 (RSM)
"OUT_116"	MD 216	REAL	// Sheet 3 (RSM)
"CNDP1"	MD 220	REAL	// Sheet 4 (RSM)
"CNDP2"	MD 224	REAL	// Sheet 4 (RSM)
"CNDP1E"	MD 228	REAL	// Sheet 4 (RSM)
"CNDP2E"	MD 232	REAL	// Sheet 4 (RSM)
"OUT_047"	MD 236	REAL	// Sheet 4 (RSM)
"OUT_048"	MD 240	REAL	// Sheet 4 (RSM)
"TICM"	MD 244	REAL	// Sheet 4 (RSM)
"FSMT1E"	MD 252	REAL	// Sheet 4 (RSM)
"FSMTAVG"	MD 256	REAL	// Sheet 4 (RSM)
"OUT_103"	MD 260	REAL	// Sheet 4 (RSM)
"OUT_104"	MD 264	REAL	// Sheet 4 (RSM)
"OUT_105"	MD 268	REAL	// Sheet 4 (RSM)
"FSMT1"	MD 272	REAL	// Sheet 4 (RSM)
"OUT_106"	MD 276	REAL	// Sheet 4 (RSM)
"Z790"	MD 280	REAL	// Sheet 4 (RSM)
"HPICOL"	MD 284	REAL	// Sheet 6 (RSM)
"ONEMINCT"	MD 288	REAL	// Sheet 6 (RSM)
"OUT_317"	MD 292	REAL	// Sheet 6 (RSM)
"IAVCT"	MD 296	REAL	// Sheet 6 (RSM)
"ISPOUTCT"	MD 300	REAL	// Sheet 6 (RSM)
"HXFER"	MD 304	REAL	// Sheet 8 (RSM)
"OUT_310"	MD 308	REAL	// Sheet 9 (RSM)
"OUT_312"	MD 312	REAL	// Sheet 9 (RSM)
"OUT_313"	MD 316	REAL	// Sheet 9 (RSM)
"OUT_311"	MD 320	REAL	// Sheet 9 (RSM)
"T6"	MD 324	REAL	// Sheet 10 (RSM)
"TP1"	MD 328	REAL	// Sheet 9 (RSM)
"TP2"	MD 332	REAL	// Sheet 9 (RSM)
"TP3"	MD 336	REAL	// Sheet 9 (RSM)
"TP4"	MD 340	REAL	// Sheet 9 (RSM)
"TP5"	MD 344	REAL	// Sheet 9 (RSM)
"T1"	MD 348	REAL	// Sheet 9 (RSM)
"T2"	MD 352	REAL	// Sheet 9 (RSM)
"T3"	MD 356	REAL	// Sheet 9 (RSM)
"T4"	MD 360	REAL	// Sheet 9 (RSM)
"T5"	MD 364	REAL	// Sheet 9 (RSM)
"ROTSURF"	MD 368	REAL	// Sheet 9 (RSM)
"OUT_315"	MD 372	REAL	// Sheet 9 (RSM)
"OUT_327"	MD 376	REAL	// Sheet 9 (RSM)
"OUT_330"	MD 380	REAL	// Sheet 9 (RSM)
"OUT_333"	MD 384	REAL	// Sheet 9 (RSM)
"OUT_336"	MD 388	REAL	// Sheet 9 (RSM)
"OUT_136"	MD 392	REAL	// Sheet 8 (RSM)
"TM1HP2"	MD 396	REAL	// Sheet 8 (RSM)
"TM2HP2"	MD 400	REAL	// Sheet 8 (RSM)
"OUT_414"	MD 404	REAL	// Sheet 8 (RSM)
"OUT_412"	MD 408	REAL	// Sheet 8 (RSM)
"OUT_413"	MD 412	REAL	// Sheet 8 (RSM)
"OUT_415"	MD 416	REAL	// Sheet 8 (RSM)
"OUT_416"	MD 420	REAL	// Sheet 8 (RSM)
"Z417"	MD 424	REAL	// Sheet 8 (RSM)
"OUT_224"	MD 428	REAL	// Sheet 8 (RSM)
"OUT_222"	MD 432	REAL	// Sheet 8 (RSM)
"TSTM"	MD 436	REAL	// Sheet 8 (RSM)
"OUT_225"	MD 440	REAL	// Sheet 8 (RSM)
"OUT_226"	MD 444	REAL	// Sheet 8 (RSM)
"TWC"	MD 448	REAL	// Sheet 8 (RSM)
"TP6"	MD 452	REAL	// Sheet 10 (RSM)
"TP7"	MD 456	REAL	// Sheet 10 (RSM)
"TP8"	MD 460	REAL	// Sheet 10 (RSM)
"TP9"	MD 464	REAL	// Sheet 10 (RSM)
"TP10"	MD 468	REAL	// Sheet 10 (RSM)
"TP11"	MD 472	REAL	// Sheet 10 (RSM)
"TP12"	MD 476	REAL	// Sheet 10 (RSM)
"TP13"	MD 480	REAL	// Sheet 10 (RSM)
"TP14"	MD 484	REAL	// Sheet 10 (RSM)
"TP15"	MD 488	REAL	// Sheet 10 (RSM)
"OUT_339"	MD 492	REAL	// Sheet 10 (RSM)
"OUT_342"	MD 496	REAL	// Sheet 10 (RSM)
"OUT_345"	MD 500	REAL	// Sheet 10 (RSM)
"OUT_348"	MD 504	REAL	// Sheet 10 (RSM)
"OUT_351"	MD 508	REAL	// Sheet 10 (RSM)
"OUT_354"	MD 512	REAL	// Sheet 10 (RSM)
"OUT_357"	MD 516	REAL	// Sheet 10 (RSM)
"OUT_360"	MD 520	REAL	// Sheet 10 (RSM)
"OUT_363"	MD 524	REAL	// Sheet 10 (RSM)
"T7"	MD 532	REAL	// Sheet 10 (RSM)
"T8"	MD 536	REAL	// Sheet 10 (RSM)
"T9"	MD 540	REAL	// Sheet 10 (RSM)
"T10"	MD 544	REAL	// Sheet 10 (RSM)
"T11"	MD 548	REAL	// Sheet 10 (RSM)
"T12"	MD 552	REAL	// Sheet 10 (RSM)
"T13"	MD 556	REAL	// Sheet 10 (RSM)
"T14"	MD 560	REAL	// Sheet 10 (RSM)
"T15"	MD 564	REAL	// Sheet 10 (RSM)
"T16"	MD 568	REAL	// Sheet 11 (RSM)
"OUT_377"	MD 572	REAL	// Sheet 10 (RSM)
"TP16"	MD 576	REAL	// Sheet 11 (RSM)
"TP17"	MD 580	REAL	// Sheet 11 (RSM)
"TP18"	MD 584	REAL	// Sheet 11 (RSM)
"TP19"	MD 588	REAL	// Sheet 11 (RSM)
"TP20"	MD 592	REAL	// Sheet 11 (RSM)
"TP21"	MD 596	REAL	// Sheet 11 (RSM)
"TP22"	MD 600	REAL	// Sheet 11 (RSM)
"TP23"	MD 604	REAL	// Sheet 11 (RSM)
"OUT_302"	MD 608	REAL	// Sheet 11 (RSM)
"OUT_305"	MD 612	REAL	// Sheet 11 (RSM)
"OUT_308"	MD 616	REAL	// Sheet 11 (RSM)
"OUT_421"	MD 620	REAL	// Sheet 11 (RSM)
"OUT_424"	MD 624	REAL	// Sheet 11 (RSM)
"OUT_427"	MD 628	REAL	// Sheet 11 (RSM)
"OUT_430"	MD 632	REAL	// Sheet 11 (RSM)
"OUT_433"	MD 636	REAL	// Sheet 11 (RSM)
"T17"	MD 640	REAL	// Sheet 11 (RSM)
"T18"	MD 644	REAL	// Sheet 11 (RSM)
"T19"	MD 648	REAL	// Sheet 11 (RSM)
"T20"	MD 652	REAL	// Sheet 11 (RSM)
"T21"	MD 656	REAL	// Sheet 11 (RSM)
"T22"	MD 660	REAL	// Sheet 11 (RSM)
"T23"	MD 664	REAL	// Sheet 11 (RSM)
"ROTBOR"	MD 668	REAL	// Sheet 11 (RSM)
"OUT_162"	MD 672	REAL	// Sheet 12 (RSM)
"OUT_163"	MD 676	REAL	// Sheet 12 (RSM)
"TNUM"	MD 680	REAL	// Sheet 12 (RSM)
"TAVG"	MD 684	REAL	// Sheet 12 (RSM)
"OUT_167"	MD 688	REAL	// Sheet 13 (RSM)
"OUT_168"	MD 692	REAL	// Sheet 13 (RSM)
"OUT_169"	MD 696	REAL	// Sheet 13 (RSM)
"HPEFFT"	MD 704	REAL	// Sheet 13 (RSM)
"HPEFFTM"	MD 708	REAL	// Sheet 13 (RSM)
"AHPEFFT"	MD 712	REAL	// Sheet 13 (RSM)
"AHPEFFTM"	MD 716	REAL	// Sheet 13 (RSM)
"OUT_170"	MD 720	REAL	// Sheet 13 (RSM)
"OUT_171"	MD 724	REAL	// Sheet 13 (RSM)
"OUT_172"	MD 728	REAL	// Sheet 13 (RSM)
"OUT_173"	MD 732	REAL	// Sheet 13 (RSM)
"OUT_174"	MD 736	REAL	// Sheet 13 (RSM)
"TDIFT2"	MD 744	REAL	// Sheet 15 (RSM)
"TDIFT3"	MD 748	REAL	// Sheet 15 (RSM)
"TDIFT4"	MD 752	REAL	// Sheet 15 (RSM)
"TDIFT5"	MD 756	REAL	// Sheet 15 (RSM)
"TDIFT6"	MD 760	REAL	// Sheet 15 (RSM)
"TDIFT7"	MD 764	REAL	// Sheet 15 (RSM)
"TDIFT8"	MD 768	REAL	// Sheet 15 (RSM)
"TDIFT9"	MD 772	REAL	// Sheet 15 (RSM)
"TDIFT10"	MD 776	REAL	// Sheet 15 (RSM)
"TDIFT11"	MD 780	REAL	// Sheet 15 (RSM)
"TDIFT12"	MD 784	REAL	// Sheet 15 (RSM)
"TDIFT13"	MD 788	REAL	// Sheet 15 (RSM)
"TDIFT14"	MD 792	REAL	// Sheet 15 (RSM)
"TDIFT15"	MD 796	REAL	// Sheet 15 (RSM)
"TDIFT1"	MD 800	REAL	// Sheet 15 (RSM)
"OUT_291"	MD 804	REAL	// Sheet 16 (RSM)
"OUT_292"	MD 808	REAL	// Sheet 16 (RSM)
"TDIFSUM"	MD 812	REAL	// Sheet 16 (RSM)
"OUT_294"	MD 816	REAL	// Sheet 16 (RSM)
"OUT_295"	MD 820	REAL	// Sheet 16 (RSM)
"ATDIF"	MD 824	REAL	// Sheet 16 (RSM)
"AATDIF"	MD 828	REAL	// Sheet 16 (RSM)
"HPRTRSLM"	MD 832	REAL	// Sheet 22 (RSM)
"VPOSL"	MD 836	REAL	// Sheet 29 (OA)
"OUT_X111"	MD 840	REAL	// Sheet 17 (RSM)
"OUT_X731"	MD 844	REAL	// Sheet 17 (RSM)
"OUT_X113"	MD 848	REAL	// Sheet 17 (RSM)
"OUT_X115"	MD 852	REAL	// Sheet 17 (RSM)
"OUT_X112"	MD 856	REAL	// Sheet 17 (RSM)
"OUT_X114"	MD 860	REAL	// Sheet 17 (RSM)
"OUT_X116"	MD 864	REAL	// Sheet 17 (RSM)
"OUT_X091"	MD 868	REAL	// Sheet 17 (RSM)
"HPRTRSL"	MD 872	REAL	// Sheet 22 (RSM)
"WSWS"	MD 876	REAL	// Sheet 18 (RSM)
"PSUM41"	MD 880	REAL	// Sheet 18 (RSM)
"PSUM42"	MD 884	REAL	// Sheet 18 (RSM)
"TTINCR"	MD 888	REAL	// Sheet 18 (RSM)
"STINCR"	MD 892	REAL	// Sheet 18 (RSM)
"TINCR"	MD 896	REAL	// Sheet 18 (RSM)
"STDECR"	MD 900	REAL	// Sheet 18 (RSM)
"TTDECR"	MD 904	REAL	// Sheet 18 (RSM)
"TDECR"	MD 908	REAL	// Sheet 18 (RSM)
"OUT_X142"	MD 912	REAL	// Sheet 18 (RSM)
"OUT_X144"	MD 920	REAL	// Sheet 18 (RSM)
"TBP"	MD 924	REAL	// Sheet 2 (RSM)
"OUT_400"	MD 928	REAL	// Sheet 20 (RSM)
"OUT_883"	MD 932	REAL	// Sheet 20 (RSM)
"OUT_882"	MD 936	REAL	// Sheet 20 (RSM)
"OUT_884"	MD 940	REAL	// Sheet 20 (RSM)
"OUT_044"	MD 944	REAL	// Sheet 20 (RSM)
"OUT_042"	MD 948	REAL	// Sheet 20 (RSM)
"OUT_885"	MD 952	REAL	// Sheet 20 (RSM)
"OUT_886"	MD 956	REAL	// Sheet 20 (RSM)
"OUT_887"	MD 960	REAL	// Sheet 20 (RSM)
"OUT_876"	MD 964	REAL	// Sheet 20 (RSM)
"MW"	MD 968	REAL	// Sheet 20 (RSM)
"OUT_875"	MD 972	REAL	// Sheet 20 (RSM)
"MWINCR"	MD 976	REAL	// Sheet 20 (RSM)
"OUT_891"	MD 980	REAL	// Sheet 20 (RSM)
"OUT_890"	MD 984	REAL	// Sheet 20 (RSM)
"OUT_889"	MD 988	REAL	// Sheet 20 (RSM)
"OUT_893"	MD 992	REAL	// Sheet 20 (RSM)
"OUT_892"	MD 996	REAL	// Sheet 20 (RSM)
"OUT_894"	MD 1000	REAL	// Sheet 20 (RSM)
"OUT_895"	MD 1004	REAL	// Sheet 20 (RSM)
"OUT_896"	MD 1008	REAL	// Sheet 20 (RSM)
"OUT_897"	MD 1012	REAL	// Sheet 20 (RSM)
"Z897"	MD 1016	REAL	// Sheet 20 (RSM)
"REFDMD"	MD 1020	REAL	// Sheet 13 (OA)
"DEMAND"	MD 1024	REAL	// Sheet 10 (OA)
"TRATELD"	MD 1028	REAL	// Sheet 46 (ATC)
"TRATEWS"	MD 1032	REAL	// Sheet 21 (RSM)
"MWDECR"	MD 1036	REAL	// Sheet 21 (RSM)
"OUT_323"	MD 1044	REAL	// Sheet 21 (RSM)
"DCLDRES"	MD 1048	REAL	// Sheet 21 (RSM)
"INLDRES"	MD 1052	REAL	// Sheet 21 (RSM)
"ATCLRAT1"	MD 1056	REAL	// Sheet 21 (RSM)
"TRATE"	MD 1060	REAL	// Sheet 21 (RSM)
"OUT_X732"	MD 1064	REAL	// Sheet 21 (RSM)
"OUT_X736"	MD 1072	REAL	// Sheet 21 (RSM)
"ATCARAT"	MD 1080	REAL	// Sheet 21 (RSM)
"OUT_577"	MD 1084	REAL	// Sheet 21 (RSM)
"OUT_159"	MD 1092	REAL	// Sheet 22 (RSM)
"HPRSLNEG"	MD 1096	REAL	// Sheet 22 (RSM)
"REFF1"	MD 1100	REAL	// Sheet 49 (ATC)
"REFF2"	MD 1104	REAL	// Sheet 49 (ATC)
"REFF3"	MD 1108	REAL	// Sheet 49 (ATC)
"REFF4"	MD 1112	REAL	// Sheet 49 (ATC)
"REFF5"	MD 1116	REAL	// Sheet 49 (ATC)
"ATCSPDRF"	MD 1120	REAL	// Sheet 30 (ATC)
"DEHDMD"	MD 1124	REAL	// Sheet 24 (RSM)
"OUT_X712"	MD 1128	REAL	// Sheet 24 (RSM)
"OUT_X715"	MD 1132	REAL	// Sheet 24 (RSM)
"OUT_X717"	MD 1136	REAL	// Sheet 24 (RSM)
"OUT_X721"	MD 1140	REAL	// Sheet 24 (RSM)
"DMDTEMP3"	MD 1144	REAL	// Sheet 24 (RSM)
"OUT_X723"	MD 1148	REAL	// Sheet 24 (RSM)
"OUT_X741"	MD 1152	REAL	// Sheet 24 (RSM)
"OUT_X701"	MD 1160	REAL	// Sheet 24 (RSM)
"OUT_X707"	MD 1164	REAL	// Sheet 24 (RSM)
"OUT_X171"	MD 1168	REAL	// Sheet 24 (RSM)
"DMDTEMP2"	MD 1172	REAL	// Sheet 24 (RSM)
"OCITE"	MD 1176	REAL	// Sheet 37 (RSM)
"OCOTE"	MD 1180	REAL	// Sheet 37 (RSM)
"OCIT"	MD 1184	REAL	// Sheet 37 (RSM)
"OCOT"	MD 1188	REAL	// Sheet 37 (RSM)
"LPGST"	MD 1192	REAL	// Sheet 7 (ATC)
"LPGSTE"	MD 1196	REAL	// Sheet 7 (ATC)
"JTBRMAL"	MD 1200	REAL	// Sheet 49 (ATC)
"BMTTLIM"	MD 1204	REAL	// Sheet 49 (ATC)
"GENBTLIM"	MD 1208	REAL	// Sheet 49 (ATC)
"GENBALIM"	MD 1212	REAL	// Sheet 49 (ATC)
"B1TH1"	MD 1228	REAL	// Sheet 12 (ATC)
"B2THI"	MD 1256	REAL	// Sheet 12 (ATC)
"B3THI"	MD 1284	REAL	// Sheet 12 (ATC)
"B7THI"	MD 1304	REAL	// Sheet 12 (ATC)
"B4THI"	MD 1308	REAL	// Sheet 12 (ATC)
"B5THI"	MD 1312	REAL	// Sheet 12 (ATC)
"B6THI"	MD 1316	REAL	// Sheet 12 (ATC)
"B10THI"	MD 1320	REAL	// Sheet 12 (ATC)
"B8THI"	MD 1324	REAL	// Sheet 12 (ATC)
"B9THI"	MD 1328	REAL	// Sheet 12 (ATC)
"TBMTTLIM"	MD 1332	REAL	// Sheet 49 (ATC)
"TTBRMAL"	MD 1336	REAL	// Sheet 49 (ATC)
"TBFCTHI"	MD 1340	REAL	// Sheet 49 (ATC)
"TBRCTHI"	MD 1344	REAL	// Sheet 49 (ATC)
"B1T1"	MD 1348	REAL	// Sheet 12 (ATC)
"OUT_GBA1"	MD 1352	REAL	// Sheet 12 (ATC)
"B1T2"	MD 1356	REAL	// Sheet 12 (ATC)
"OUT_GBA2"	MD 1360	REAL	// Sheet 12 (ATC)
"B2T1"	MD 1364	REAL	// Sheet 12 (ATC)
"B2T2"	MD 1368	REAL	// Sheet 12 (ATC)
"B3T1"	MD 1372	REAL	// Sheet 12 (ATC)
"B3T2"	MD 1376	REAL	// Sheet 12 (ATC)
"B4T1"	MD 1384	REAL	// Sheet 12 (ATC)
"B4T2"	MD 1388	REAL	// Sheet 12 (ATC)
"B5T1"	MD 1392	REAL	// Sheet 12 (ATC)
"B5T2"	MD 1396	REAL	// Sheet 12 (ATC)
"B6T1"	MD 1400	REAL	// Sheet 12 (ATC)
"B6T2"	MD 1404	REAL	// Sheet 12 (ATC)
"B10T"	MD 1408	REAL	// Sheet 12 (ATC)
"B8T"	MD 1412	REAL	// Sheet 12 (ATC)
"B9T"	MD 1416	REAL	// Sheet 12 (ATC)
"TBFLT1"	MD 1420	REAL	// Sheet 12 (ATC)
"TBFLT2"	MD 1424	REAL	// Sheet 12 (ATC)
"TBFCT1"	MD 1428	REAL	// Sheet 12 (ATC)
"TBFCT2"	MD 1432	REAL	// Sheet 12 (ATC)
"TBRCT1"	MD 1436	REAL	// Sheet 12 (ATC)
"TBRCT2"	MD 1440	REAL	// Sheet 12 (ATC)
"TBRLT1"	MD 1444	REAL	// Sheet 12 (ATC)
"TBRLT2"	MD 1448	REAL	// Sheet 12 (ATC)
"OUT_GBA3"	MD 1452	REAL	// Sheet 12 (ATC)
"OUT_GBA4"	MD 1456	REAL	// Sheet 12 (ATC)
"OUT_GBA5"	MD 1460	REAL	// Sheet 12 (ATC)
"OUT_GBA6"	MD 1464	REAL	// Sheet 12 (ATC)
"OUT_GBA7"	MD 1468	REAL	// Sheet 12 (ATC)
"OUT_GBA8"	MD 1472	REAL	// Sheet 12 (ATC)
"OUT_GBA9"	MD 1476	REAL	// Sheet 12 (ATC)
"OUT_GBA10"	MD 1480	REAL	// Sheet 12 (ATC)
"OUT_GBA11"	MD 1484	REAL	// Sheet 12 (ATC)
"OUT_GBA12"	MD 1488	REAL	// Sheet 12 (ATC)
"OUT_GBA13"	MD 1492	REAL	// Sheet 12 (ATC)
"OUT_GBA14"	MD 1496	REAL	// Sheet 12 (ATC)
"OUT_GBA15"	MD 1500	REAL	// Sheet 12 (ATC)
"OUT_GBA16"	MD 1504	REAL	// Sheet 12 (ATC)
"TBFLTA1"	MD 1508	REAL	// Sheet 12 (ATC)
"TBFLTA2"	MD 1512	REAL	// Sheet 12 (ATC)
"TBFCTA1"	MD 1516	REAL	// Sheet 12 (ATC)
"TBFCTA2"	MD 1520	REAL	// Sheet 12 (ATC)
"TBRCTA1"	MD 1524	REAL	// Sheet 12 (ATC)
"TBRCTA2"	MD 1528	REAL	// Sheet 12 (ATC)
"TBRLTA1"	MD 1532	REAL	// Sheet 12 (ATC)
"TBRLTA2"	MD 1536	REAL	// Sheet 12 (ATC)
"RPCNTR"	MD 1540	REAL	// Sheet 49 (ATC)
"RPALRM1"	MD 1544	REAL	// Sheet 49 (ATC)
"A50"	MD 1548	REAL	// Sheet 48 (ATC)
"RPTRIP1"	MD 1552	REAL	// Sheet 49 (ATC)
"RPALRM5"	MD 1556	REAL	// Sheet 49 (ATC)
"RPTRIP5"	MD 1560	REAL	// Sheet 49 (ATC)
"DEALRM2"	MD 1564	REAL	// Sheet 49 (ATC)
"DEALRM1"	MD 1568	REAL	// Sheet 49 (ATC)
"DETRIP2"	MD 1572	REAL	// Sheet 49 (ATC)
"DETRIP1"	MD 1576	REAL	// Sheet 49 (ATC)
"RP1"	MD 1580	REAL	// Sheet 15 (ATC)
"RP2"	MD 1584	REAL	// Sheet 15 (ATC)
"DEGEN"	MD 1588	REAL	// Sheet 15 (ATC)
"OUT_GBA25"	MD 1592	REAL	// Sheet 15 (ATC)
"OUT_GBA26"	MD 1596	REAL	// Sheet 15 (ATC)
"OUT_GBA27"	MD 1600	REAL	// Sheet 15 (ATC)
"OUT_A413"	MD 1604	REAL	// Sheet 15 (ATC)
"OUT_407"	MD 1608	REAL	// Sheet 15 (ATC)
"OUT_408"	MD 1612	REAL	// Sheet 15 (ATC)
"OUT_A414"	MD 1616	REAL	// Sheet 15 (ATC)
"DEGENR"	MD 1620	REAL	// Sheet 15 (ATC)
"OUT_X431"	MD 1624	REAL	// Sheet 15 (ATC)
"RPOS"	MD 1628	REAL	// Sheet 15 (ATC)
"RATELD"	MD 1632	REAL	// Sheet 49 (ATC)
"OUT_129"	MD 1636	REAL	// Sheet 17 (ATC)
"CNDLIMS"	MD 1640	REAL	// Sheet 17 (ATC)
"CNDLIMMW"	MD 1644	REAL	// Sheet 17 (ATC)
"OUT_A882"	MD 1648	REAL	// Sheet 17 (ATC)
"OUT_A883"	MD 1652	REAL	// Sheet 17 (ATC)
"OUT_A136"	MD 1656	REAL	// Sheet 17 (ATC)
"OUT_127"	MD 1660	REAL	// Sheet 17 (ATC)
"INHG"	MD 1664	REAL	// Sheet 17 (ATC)
"LP1GVT"	MD 1668	REAL	// Sheet 17 (ATC)
"LP2GVT"	MD 1672	REAL	// Sheet 17 (ATC)
"LP1GNT"	MD 1676	REAL	// Sheet 17 (ATC)
"LP2GNT"	MD 1680	REAL	// Sheet 17 (ATC)
"OUT_GBA28"	MD 1684	REAL	// Sheet 17 (ATC)
"OUT_GBA29"	MD 1688	REAL	// Sheet 17 (ATC)
"OUT_GBA30"	MD 1692	REAL	// Sheet 17 (ATC)
"OUT_GBA31"	MD 1696	REAL	// Sheet 17 (ATC)
"LPEXSTHI"	MD 1700	REAL	// Sheet 17 (ATC)
"OUT_233A"	MD 1704	REAL	// Supporting variable in sheet 17 (ATC)
"OUT_233B"	MD 1708	REAL	// Supporting variable in sheet 17 (ATC)
"EIGHT"	MD 1712	REAL	// Sheet 48 (ATC)
"FIVE"	MD 1716	REAL	// Sheet 48 (ATC)
"NINE"	MD 1720	REAL	// Sheet 48 (ATC)
"SIX"	MD 1724	REAL	// Sheet 48 (ATC)
"THREE"	MD 1728	REAL	// Sheet 48 (ATC)
"TWO"	MD 1732	REAL	// Sheet 48 (ATC)
"OUT_600"	MD 1736	REAL	// Sheet 20 (ATC)
"OUT_618"	MD 1740	REAL	// Sheet 20 (ATC)
"VIBLIMIT"	MD 1744	REAL	// Sheet 20 (ATC)
"VIBTRIPE"	MD 1748	REAL	// Sheet 20 (ATC)
"VIBLIME"	MD 1752	REAL	// Sheet 20 (ATC)
"OUT_686"	MD 1756	REAL	// Sheet 25 (ATC)
"OUT_685"	MD 1760	REAL	// Sheet 25 (ATC)
"RPM1"	MD 1764	REAL	// Sheet 7 (OA)
"RPMM1"	MD 1768	REAL	// Sheet 7 (OA)
"RPM2"	MD 1772	REAL	// Sheet 7 (OA)
"RPM3"	MD 1776	REAL	// Sheet 7 (OA)
"RPMM3"	MD 1780	REAL	// Sheet 7 (OA)
"RPM4"	MD 1784	REAL	// Sheet 7 (OA)
"RPMM4"	MD 1788	REAL	// Sheet 7 (OA)
"RPM5"	MD 1792	REAL	// Sheet 7 (OA)
"RPMM5"	MD 1796	REAL	// Sheet 7 (OA)
"RDSPDREF"	MD 1800	REAL	// Sheet 25 (ATC)
"RUSPDREF"	MD 1804	REAL	// Sheet 25 (ATC)
"RPMM2"	MD 1808	REAL	// Sheet 7 (OA)
"EXCREFF"	MD 1812	REAL	// Sheet 49 (ATC)
"RBSPDREF"	MD 1816	REAL	// Sheet 27 (ATC)
"OUT_670"	MD 1820	REAL	// Sheet 27 (ATC)
"OUT_671"	MD 1824	REAL	// Sheet 27 (ATC)
"OUT_672"	MD 1828	REAL	// Sheet 27 (ATC)
"OUT_673"	MD 1832	REAL	// Sheet 27 (ATC)
"OUT_674"	MD 1836	REAL	// Sheet 27 (ATC)
"RPMM110"	MD 1840	REAL	// Sheet 29 (ATC)
"RPMM210"	MD 1844	REAL	// Sheet 29 (ATC)
"RPMM310"	MD 1848	REAL	// Sheet 29 (ATC)
"RPMM410"	MD 1852	REAL	// Sheet 29 (ATC)
"RPMM510"	MD 1856	REAL	// Sheet 29 (ATC)
"RPMMEX10"	MD 1860	REAL	// Sheet 29 (ATC)
"OUT_677"	MD 1864	REAL	// Sheet 29 (ATC)
"OUT_678"	MD 1868	REAL	// Sheet 29 (ATC)
"OUT_679"	MD 1872	REAL	// Sheet 29 (ATC)
"OUT_680"	MD 1876	REAL	// Sheet 29 (ATC)
"OUT_681"	MD 1880	REAL	// Sheet 29 (ATC)
"RTSPDREF"	MD 1884	REAL	// Sheet 29 (ATC)
"OUT_900"	MD 1888	REAL	// Sheet 30 (ATC)
"OUT_684"	MD 1892	REAL	// Sheet 30 (ATC)
"HLDSPDRF"	MD 1896	REAL	// Sheet 30 (ATC)
"OUT_691"	MD 1900	REAL	// Sheet 30 (ATC)
"Z995"	MD 1908	REAL	// Sheet 30 (ATC)
"OUT_693"	MD 1912	REAL	// Sheet 30 (ATC)
"OUT_694"	MD 1916	REAL	// Sheet 30 (ATC)
"OUT_687"	MD 1920	REAL	// Sheet 30 (ATC)
"OUT_688"	MD 1924	REAL	// Sheet 30 (ATC)
"OUT_689"	MD 1928	REAL	// Sheet 30 (ATC)
"OUT_690"	MD 1932	REAL	// Sheet 30 (ATC)
"ATCREFLO"	MD 1936	REAL
"MWPERCT"	MD 1940	REAL	// Sheet 2 (OPC)
"LDHPDRV"	MD 1944	REAL	// Sheet 49 (ATC)
"HPBMIDT"	MD 1948	REAL	// Sheet 31 (ATC)
"HPCMIDT"	MD 1952	REAL	// Sheet 31 (ATC)
"HPBMIDTE"	MD 1956	REAL	// Sheet 31 (ATC)
"HPCMIDTE"	MD 1960	REAL	// Sheet 31 (ATC)
"OUT_X191"	MD 1964	REAL	// Sheet 31 (ATC)
"HOLDCMB"	MD 1968	REAL	// Sheet 49 (ATC)
"TRIPCMB"	MD 1972	REAL	// Sheet 49 (ATC)
"VB1"	MD 1976	REAL	// Sheet 24 (ATC)
"VB2"	MD 1980	REAL	// Sheet 24 (ATC)
"VB3"	MD 1984	REAL	// Sheet 24 (ATC)
"VB4"	MD 1988	REAL	// Sheet 24 (ATC)
"VB5"	MD 1992	REAL	// Sheet 24 (ATC)
"VB6"	MD 1996	REAL	// Sheet 24 (ATC)
"VB7"	MD 2000	REAL	// Sheet 24 (ATC)
"VB8"	MD 2004	REAL	// Sheet 24 (ATC)
"VB9"	MD 2008	REAL	// Sheet 24 (ATC)
"VB10"	MD 2012	REAL	// Sheet 24 (ATC)
"VBA1"	MD 2016	REAL	// Sheet 24 (ATC)
"VBA2"	MD 2020	REAL	// Sheet 24 (ATC)
"VBA3"	MD 2024	REAL	// Sheet 24 (ATC)
"VBA4"	MD 2028	REAL	// Sheet 24 (ATC)
"VBA5"	MD 2032	REAL	// Sheet 24 (ATC)
"VBA6"	MD 2036	REAL	// Sheet 24 (ATC)
"VBA7"	MD 2040	REAL	// Sheet 24 (ATC)
"VBA8"	MD 2044	REAL	// Sheet 24 (ATC)
"VBA9"	MD 2048	REAL	// Sheet 24 (ATC)
"VBA10"	MD 2052	REAL	// Sheet 24 (ATC)
"VIBTRIP"	MD 2056	REAL	// Sheet 24 (ATC)
"EHFLT"	MD 2060	REAL	// Sheet 33 (ATC)
"EHFLTE"	MD 2064	REAL	// Sheet 33 (ATC)
"OUT_X601"	MD 2068	REAL	// Sheet 35 (ATC)
"OUT_X602"	MD 2072	REAL	// Sheet 35 (ATC)
"OUT_998"	MD 2076	REAL	// Sheet 35 (ATC)
"OUT_997"	MD 2080	REAL	// Sheet 35 (ATC)
"OUT_996"	MD 2084	REAL	// Sheet 35 (ATC)
"OUT_999"	MD 2088	REAL	// Sheet 35 (ATC)
"ROTECCE"	MD 2092	REAL	// Sheet 35 (ATC)
"OUT_X222"	MD 2096	REAL	// Sheet 35 (ATC)
"TBRLTAVG"	MD 2100	REAL	// Sheet 35 (ATC)
"TBFRTAVG"	MD 2104	REAL	// Sheet 35 (ATC)
"TBRCTAVG"	MD 2108	REAL	// Sheet 35 (ATC)
"TBFTAVG"	MD 2112	REAL	// Sheet 35 (ATC)
"OUT_A312"	MD 2116	REAL	// Sheet 35 (ATC)
"OUT_314"	MD 2120	REAL	// Sheet 35 (ATC)
"OUT_316"	MD 2124	REAL	// Sheet 35 (ATC)
"OUT_318"	MD 2128	REAL	// Sheet 35 (ATC)
"ROTECC"	MD 2132	REAL	// Sheet 35 (ATC)
"OUT_X652"	MD 2136	REAL	// Sheet 46 (ATC)
"OUT_X654"	MD 2140	REAL	// Sheet 46 (ATC)
"OUT_X656"	MD 2144	REAL	// Sheet 46 (ATC)
"RATIDX"	MD 2148	REAL	// Sheet 46 (ATC)
"RATEINDX"	MD 2152	REAL	// Sheet 46 (ATC)
"OUT_X631"	MD 2156	REAL	// Sheet 46 (ATC)
"OUT_X633"	MD 2160	REAL	// Sheet 46 (ATC)
"OUT_X635"	MD 2164	REAL	// Sheet 46 (ATC)
"RATETEMP"	MD 2172	REAL	// Sheet 46 (ATC)
"OUT_X638"	MD 2176	REAL	// Sheet 46 (ATC)
"OUT_X651"	MD 2180	REAL	// Sheet 46 (ATC)
"PRCHPT1"	MD 2184	REAL	// Sheet 48 (ATC)
"PRCHKPT2"	MD 2188	REAL	// Sheet 48 (ATC)
"R21"	MD 2192	REAL	// Sheet 48 (ATC)
"R11"	MD 2196	REAL	// Sheet 48 (ATC)
"R31"	MD 2200	REAL	// Sheet 48 (ATC)
"R22"	MD 2204	REAL	// Sheet 48 (ATC)
"R32"	MD 2208	REAL	// Sheet 48 (ATC)
"R23"	MD 2212	REAL	// Sheet 48 (ATC)
"R13"	MD 2216	REAL	// Sheet 48 (ATC)
"R33"	MD 2220	REAL	// Sheet 48 (ATC)
"XP921"	MD 2224	REAL	// Sheet 48 (ATC)
"XP911"	MD 2228	REAL	// Sheet 48 (ATC)
"XP931"	MD 2232	REAL	// Sheet 48 (ATC)
"XP922"	MD 2236	REAL	// Sheet 48 (ATC)
"XP912"	MD 2240	REAL	// Sheet 48 (ATC)
"XP932"	MD 2244	REAL	// Sheet 48 (ATC)
"YP922"	MD 2248	REAL	// Sheet 48 (ATC)
"YP912"	MD 2252	REAL	// Sheet 48 (ATC)
"YP932"	MD 2256	REAL	// Sheet 48 (ATC)
"XP923"	MD 2260	REAL	// Sheet 48 (ATC)
"XP913"	MD 2264	REAL	// Sheet 48 (ATC)
"XP933"	MD 2268	REAL	// Sheet 48 (ATC)
"YP923"	MD 2272	REAL	// Sheet 48 (ATC)
"YP913"	MD 2276	REAL	// Sheet 48 (ATC)
"YP933"	MD 2280	REAL	// Sheet 48 (ATC)
"R12"	MD 2284	REAL	// Sheet 48 (ATC)
"YP921"	MD 2288	REAL	// Sheet 48 (ATC)
"YP911"	MD 2292	REAL	// Sheet 48 (ATC)
"YP931"	MD 2296	REAL	// Sheet 48 (ATC)
"Z275"	MW 740	INT	// Sheet 14 (RSM)
"Z036"	MW 1216	INT	// Sheet 3 (ATC)
"Main program routine"	OB 1	OB 1
"I/O_FLT1"	OB 82	OB 82	// I/O Point Fault 1
"I/O_FLT2"	OB 83	OB 83	// I/O Point Fault 2
"OBNL_FLT"	OB 85	OB 85	// OB Not Loaded Fault
"RACK_FLT"	OB 86	OB 86	// Loss of Rack Fault
"COMPLETE RESTART"	OB 100	OB 100	// Complete Restart
"PROG_ERR"	OB 121	OB 121	// Programming Error
"MOD_ERR"	OB 122	OB 122	// Module Access Error
"ATCALO"	Q 0.0	BOOL	//  (ATC) - (FieldIO4-M2)
"ATCASSO"	Q 0.1	BOOL	//  (ATC) - (FieldIO4-M2)
"ATCMEO"	Q 0.2	BOOL	//  (ATC) - (FieldIO4-M2)
"ATCNAO"	Q 0.3	BOOL	//  (ATC) - (FieldIO4-M2)
"ATCSMO"	Q 0.4	BOOL	//  (ATC) - (FieldIO4-M2)
"ATCTAO"	Q 0.5	BOOL	//  (ATC) - (FieldIO4-M2)
"ATCTO"	Q 0.6	BOOL	//  (ATC) - (FieldIO4-M2)
"CHPDVO"	Q 0.7	BOOL	//  (ATC) - (FieldIO4-M2)
"CRSBO"	Q 1.0	BOOL	//  (ATC) - (FieldIO4-M2)
"LPHTO"	Q 1.1	BOOL	//  (ATC) - (FieldIO4-M2)
"LPVHTO"	Q 1.2	BOOL	//  (ATC) - (FieldIO4-M2)
"WDHTO"	Q 1.3	BOOL	//  (ATC) - (FieldIO4-M2)
"WDVHTO"	Q 1.4	BOOL	//  (ATC) - (FieldIO4-M2)
"RSINV1"	Q 2.0	BOOL	//  (RSM) - (FieldIO5-M2)
"RSINV2"	Q 2.1	BOOL	//  (RSM) - (FieldIO5-M2)
"RSMON1"	Q 2.2	BOOL	//  (RSM) - (FieldIO5-M2)
"RSMON2"	Q 2.3	BOOL	//  (RSM) - (FieldIO5-M2)
"RSSENO"	Q 2.4	BOOL	//  (RSM) - (FieldIO5-M2)
"SPHLD"	Q 2.5	BOOL	//  (RSM) - (FieldIO5-M2)
"READ_CLK"	SFC 1	SFC 1	// Read System Clock
"TIME_TCK"	SFC 64	SFC 64	// Read the System Time
"HISIGMTR-UDT"	UDT 1	UDT 1
"LOSIGMTR-UDT"	UDT 2	UDT 2
"DBEQUALS-UDT"	UDT 3	UDT 3
"GAINBI-UDT"	UDT 4	UDT 4
"DELTAW-UDT"	UDT 5	UDT 5
"HILOLMTV-UDT"	UDT 6	UDT 6	// constants for HILOLMTV
"HILOMTR-UDT"	UDT 7	UDT 7
"HISIGMTV-UDT"	UDT 8	UDT 8
"LOSIGMTV-UDT"	UDT 9	UDT 9
"XLIMIT-UDT"	UDT 10	UDT 10
"MULTGB-UDT"	UDT 11	UDT 11
"SUM2W-UDT"	UDT 12	UDT 12
"RATEMTR-UDT"	UDT 13	UDT 13
"XSUM-UDT"	UDT 14	UDT 14
"XTRANSF-UDT"	UDT 15	UDT 15
"XHISEL_UDT"	UDT 16	UDT 16
"TRKHOLD-UDT"	UDT 18	UDT 18
"SUM4W-UDT"	UDT 20	UDT 20
"AIFCTGEN_UDT"	UDT 21	UDT 21
"DIVIDEGB_UDT"	UDT 22	UDT 22
"POLY_UDT"	UDT 23	UDT 23
"SUM8W_UDT"	UDT 24	UDT 24
"RESETSUM_UDT"	UDT 25	UDT 25
"XMULT_UDT"	UDT 26	UDT 26
"DIGCNTNF_UDT"	UDT 27	UDT 27
"TIMECHG_UDT"	UDT 28	UDT 28
END_SYMBOL_TABLE

TYPE "HISIGMTR-UDT"	// UDT 1
AUTHOR : Sabeeh
VERSION : 0.0
  STRUCT 	// Type Description
   STPT : REAL ;
   DBAN : REAL ;
  END_STRUCT ;	
END_TYPE

TYPE "LOSIGMTR-UDT"	// UDT 2
AUTHOR : Sabeeh
VERSION : 0.0
  STRUCT 	// Type Description
   STPT : REAL ;
   DBAN : REAL ;
  END_STRUCT ;	
END_TYPE

TYPE "DBEQUALS-UDT"	// UDT 3
AUTHOR : Sabeeh
VERSION : 0.0
  STRUCT 	// Type Description
   DBAN : REAL ;
   RTRN : REAL ;
  END_STRUCT ;	
END_TYPE

TYPE "GAINBI-UDT"	// UDT 4
AUTHOR : Sabeeh
VERSION : 0.0
  STRUCT 	// Type Description
   GAIN : REAL ;
   BIAS : REAL ;
  END_STRUCT ;	
END_TYPE

TYPE "DELTAW-UDT"	// UDT 5
AUTHOR : Sabeeh
VERSION : 0.0
  STRUCT 	// Type Description
   WT1 : REAL ;
   WT2 : REAL ;
  END_STRUCT ;	
END_TYPE

TYPE "HILOLMTV-UDT"	// UDT 6
AUTHOR : Sabeeh
VERSION : 0.0
  STRUCT 	// Type Description
   LOLM : REAL ;
   HILM : REAL ;
  END_STRUCT ;	
END_TYPE

TYPE "HILOMTR-UDT"	// UDT 7
AUTHOR : Sabeeh
VERSION : 0.0
  STRUCT 	// Type Description
   HISP : REAL ;
   HIDB : REAL ;
   LOSP : REAL ;
   LODB : REAL ;
  END_STRUCT ;	
END_TYPE

TYPE "HISIGMTV-UDT"	// UDT 8
AUTHOR : Sabeeh
VERSION : 0.0
  STRUCT 	// Type Description
   DBAN : REAL ;
  END_STRUCT ;	
END_TYPE

TYPE "LOSIGMTV-UDT"	// UDT 9
AUTHOR : Sabeeh
VERSION : 0.0
  STRUCT 	// Type Description
   DBAN : REAL ;
  END_STRUCT ;	
END_TYPE

TYPE "XLIMIT-UDT"	// UDT 10
AUTHOR : Sabeeh
VERSION : 0.0
  STRUCT 	// Type Description
   GAIN : REAL  := 1.000000e+000;
   BIAS : REAL ;
   SCLTOP : REAL  := 1.000000e+002;
   SCLBTM : REAL  := -1.000000e+002;
  END_STRUCT ;	
END_TYPE

TYPE "MULTGB-UDT"	// UDT 11
AUTHOR : Sabeeh
VERSION : 0.0
  STRUCT 	// Type Description
   GAIN : REAL ;
   BIAS : REAL ;
  END_STRUCT ;	
END_TYPE

TYPE "SUM2W-UDT"	// UDT 12
AUTHOR : Sabeeh
VERSION : 0.0
  STRUCT 	// Type Description
   WT1 : REAL ;
   WT2 : REAL ;
  END_STRUCT ;	
END_TYPE

TYPE "RATEMTR-UDT"	// UDT 13
AUTHOR : RJ
VERSION : 0.0
  STRUCT 	// Type Description
   OLDIN : REAL ;
   OLDT : TIME ;
   i : INT ;
   PRATE : REAL ;
   NRATE : REAL ;
   PDB : REAL ;
   NDB : REAL ;
  END_STRUCT ;	
END_TYPE

TYPE "XSUM-UDT"	// UDT 14
AUTHOR : Sabeeh
VERSION : 0.0
  STRUCT 	// Type Description
   PVGAIN : REAL ;
   PVBIAS : REAL ;
   CASGAIN : REAL ;
   CASBIAS : REAL ;
   SCALETOP : REAL ;
   SCALEBOT : REAL ;
  END_STRUCT ;	
END_TYPE

TYPE "XTRANSF-UDT"	// UDT 15
AUTHOR : Sabeeh
VERSION : 0.0
  STRUCT 	// Type Description
   PV_YGAIN : REAL ;
   PV_YBIAS : REAL ;
   CAS_NGAIN : REAL ;
   CAS_NBIAS : REAL ;
   SCALETOP : REAL ;
   SCALEBOT : REAL ;
  END_STRUCT ;	
END_TYPE

TYPE "XHISEL_UDT"	// UDT 16
VERSION : 0.0
  STRUCT
   PV_GAIN : REAL ;
   PV_BIAS : REAL ;
   CAS_GAIN : REAL ;
   CAS_BIAS : REAL ;
   SCALE_TOP : REAL ;
   SCALE_BOT : REAL ;
  END_STRUCT ;	
END_TYPE

TYPE "TRKHOLD-UDT"	// UDT 18
AUTHOR : Sabeeh
VERSION : 0.0
  STRUCT 	// Type Description
   temp : BOOL ;
  END_STRUCT ;	
END_TYPE

TYPE "SUM4W-UDT"	// UDT 20
AUTHOR : Sabeeh
VERSION : 0.0
  STRUCT 	// Type Description
   WT1 : REAL ;
   WT2 : REAL ;
   WT3 : REAL ;
   WT4 : REAL ;
  END_STRUCT ;	
END_TYPE

TYPE "AIFCTGEN_UDT"	// UDT 21
VERSION : 0.0
  STRUCT
   R : ARRAY  [1 .. 9 ] OF REAL ;
   S : ARRAY  [1 .. 9 ] OF REAL ;
   NMBP : INT ;
  END_STRUCT ;	
END_TYPE

TYPE "DIVIDEGB_UDT"	// UDT 22
AUTHOR : RJ
VERSION : 0.0
  STRUCT
   GAIN : REAL ;
   BIAS : REAL ;
  END_STRUCT ;	
END_TYPE

TYPE "POLY_UDT"	// UDT 23
AUTHOR : RJ
VERSION : 0.0
  STRUCT
   CX0 : REAL ;
   CX1 : REAL ;
   CX2 : REAL ;
   CX3 : REAL ;
   CX4 : REAL ;
   CX5 : REAL ;
  END_STRUCT ;	
END_TYPE

TYPE "SUM8W_UDT"	// UDT 24
AUTHOR : RJ
VERSION : 0.0
  STRUCT 	// Type Description
   WT1 : REAL ;
   WT2 : REAL ;
   WT3 : REAL ;
   WT4 : REAL ;
   WT5 : REAL ;
   WT6 : REAL ;
   WT7 : REAL ;
   WT8 : REAL ;
  END_STRUCT ;	
END_TYPE

TYPE "RESETSUM_UDT"	// UDT 25
AUTHOR : RJ
VERSION : 0.0
  STRUCT
   RCNT : REAL ;
   GAIN : REAL ;
   TRST : REAL ;
  END_STRUCT ;	
END_TYPE

TYPE "XMULT_UDT"	// UDT 26
AUTHOR : RJ
VERSION : 0.0
  STRUCT
   PV_GAIN : REAL ;
   PV_BIAS : REAL ;
   CAS_GAIN : REAL ;
   CAS_BIAS : REAL ;
   SCALE_TOP : REAL ;
   SCALE_BOT : REAL ;
  END_STRUCT ;	
END_TYPE

TYPE "DIGCNTNF_UDT"	// UDT 27
AUTHOR : RJ
VERSION : 0.0
  STRUCT
   N : INT ;
   M : INT ;
  END_STRUCT ;	
END_TYPE

TYPE "TIMECHG_UDT"	// UDT 28
AUTHOR : RJ
VERSION : 0.1
  STRUCT
   OLDH : INT ;
   OLDM : INT ;
   OLDS : INT ;
   PTIME : S5TIME ;
  END_STRUCT ;	
END_TYPE

FUNCTION_BLOCK "AIN"	// FB 1
TITLE = Scaling and Conversion of Analog Input (Words)
AUTHOR : RJ
VERSION : 0.1
VAR_INPUT
  IN : WORD ;	//Analog Input (Word)
END_VAR
VAR_OUTPUT
  OUT : REAL ;	//Output Value (Real)
END_VAR
VAR
  HIGH : REAL ;	//Upper limit
  LOW : REAL ;	//Lower limit
  BIPOLAR : BOOL ;	//Unipolar or bipolar conversion
  ERROR : WORD ;	//Range overflow error
  AI_INT : INT ;	//Analog Input (INT)
END_VAR
BEGIN
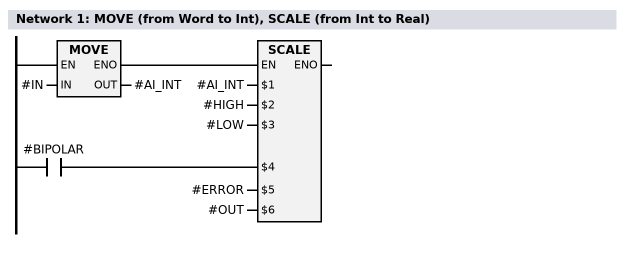
NETWORK
TITLE = MOVE (from Word to Int), SCALE (from Int to Real) 
      A     #BIPOLAR;
      =     L 0.0;
      BLD   103;
      A(;
      L     #IN;
      T     #AI_INT;
      SET;
      SAVE;
      CLR;
      A     BR;
      );
      JNB   _001;
      CALL  "SCALE" (
           $1                       := #AI_INT,
           $2                       := #HIGH,
           $3                       := #LOW,
           $4                       := L 0.0,
           $5                       := #ERROR,
           $6                       := #OUT);
_001: NOP   0;
END_FUNCTION_BLOCK

FUNCTION_BLOCK "RUNAVG"	// FB 2
AUTHOR : RJ
VERSION : 0.0
VAR_INPUT
  IN : REAL ;
END_VAR
VAR_OUTPUT
  OUT : REAL ;
END_VAR
VAR
  S_Time : DINT ;	//Time after which a sample of input is taken (Parameter)
  Time_Unit : INT ;	//Unit of time (Parameter)
  Number_Samples : INT ;	//Number of samples taken for average (Parameter)
  Sample_Time : DINT ;	//S_Time in ms
  Vector_Samples : ARRAY  [0 .. 7 ] OF //Vector containing input samples
  REAL  := 0.000000e+000, 0.000000e+000, 0.000000e+000, 0.000000e+000, 0.000000e+000, 0.000000e+000, 0.000000e+000, 0.000000e+000;	//Vector containing input samples
  Cycle_Number : INT  := 1;	//Current execution cycle of the function
  i : INT ;	//Loop variable
  OLDT : TIME ;	//Record of time
END_VAR
VAR_TEMP
  Temp_AVG : REAL ;
  NEWT : TIME ;
  TIME_ELAPSED : DINT ;
END_VAR
BEGIN
// body was compiled from an SCL source; compiled code not shown
END_FUNCTION_BLOCK

FUNCTION_BLOCK "DRUMD16"	// FB 3
AUTHOR : RJ
VERSION : 0.0
VAR_INPUT
  INC : BOOL ;
  DEC : BOOL ;
  TMOD : BOOL ;
  TRIN : REAL ;
END_VAR
VAR_OUTPUT
  STEP : INT ;
  OUT1 : BOOL ;
  OUT2 : BOOL ;
  OUT3 : BOOL ;
  OUT4 : BOOL ;
  OUT5 : BOOL ;
  OUT6 : BOOL ;
  OUT7 : BOOL ;
  OUT8 : BOOL ;
  OUT9 : BOOL ;
  OUT10 : BOOL ;
  OUT11 : BOOL ;
  OUT12 : BOOL ;
  OUT13 : BOOL ;
  OUT14 : BOOL ;
  OUT15 : BOOL ;
  OUT16 : BOOL ;
END_VAR
VAR
  IN : ARRAY  [1 .. 50 ] OF WORD ;
  NMIN : INT ;
  INC_PREV : BOOL ;
  DEC_PREV : BOOL ;
  OUT : ARRAY  [1 .. 16 ] OF BOOL ;
END_VAR
VAR_TEMP
  i : INT ;
  MASK : INT ;
END_VAR
BEGIN
// body was compiled from an SCL source; compiled code not shown
END_FUNCTION_BLOCK

FUNCTION "QC" : VOID	// FC 1
AUTHOR : RJ
VERSION : 0.1
VAR_INPUT
  IN : REAL ;
END_VAR
VAR_OUTPUT
  OUT : BOOL ;	//QCHK1BAD
END_VAR
BEGIN
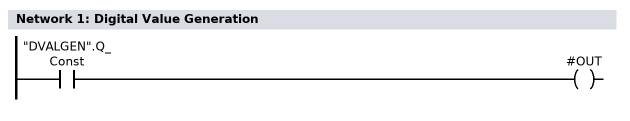
NETWORK
TITLE = Digital Value Generation
      A     "DVALGEN".Q_Const;
      =     #OUT;
END_FUNCTION

FUNCTION "Sheet 24 (ATC)" : VOID	// FC 2
TITLE = Sheet 24 (ATC)
//VIBRATION MONITOR
AUTHOR : RJ
FAMILY : ATC
VERSION : 0.1
BEGIN
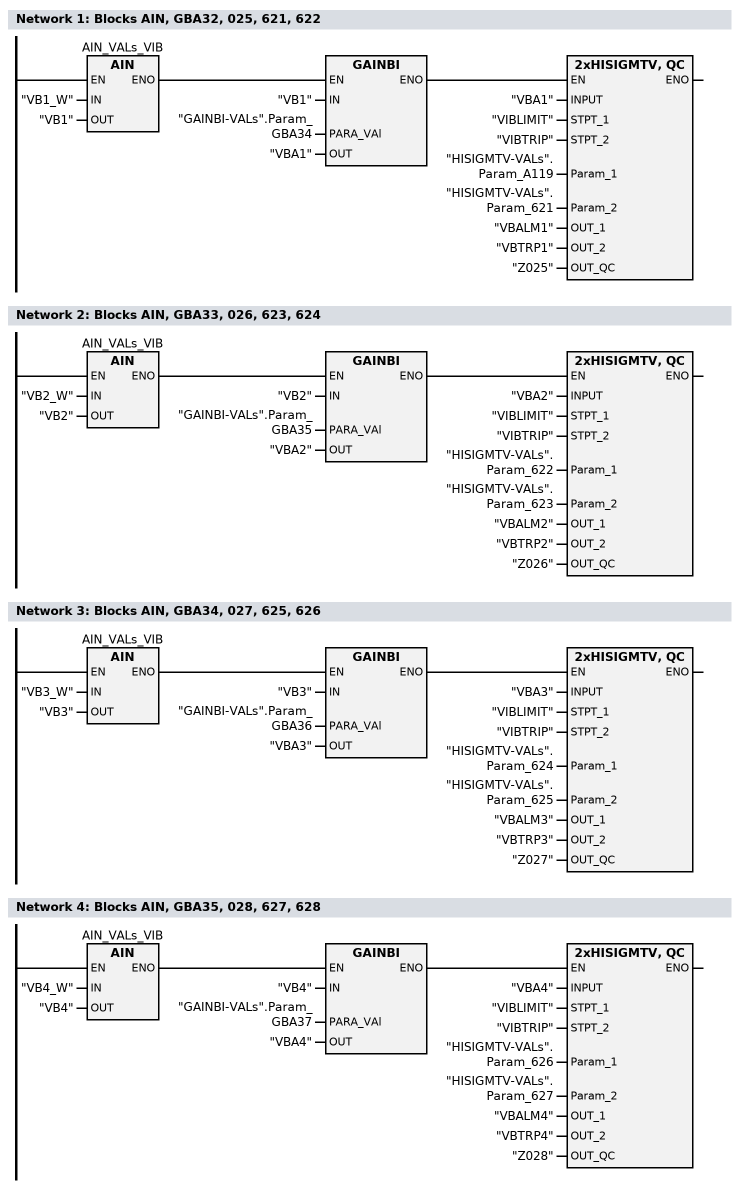
NETWORK
TITLE = Blocks AIN, GBA32, 025, 621, 622
      A(;
      A(;
      CALL  "AIN" , "AIN_VALs_VIB" (
           IN                       := "VB1_W",
           OUT                      := "VB1");
      A     BR;
      );
      JNB   _001;
      CALL  "GAINBI" (
           IN                       := "VB1",
           PARA_VAl                 := "GAINBI-VALs".Param_GBA34,
           OUT                      := "VBA1");
_001: A     BR;
      );
      JNB   _002;
      CALL  "2xHISIGMTV, QC" (
           INPUT                    := "VBA1",
           STPT_1                   := "VIBLIMIT",
           STPT_2                   := "VIBTRIP",
           Param_1                  := "HISIGMTV-VALs".Param_A119,
           Param_2                  := "HISIGMTV-VALs".Param_621,
           OUT_1                    := "VBALM1",
           OUT_2                    := "VBTRP1",
           OUT_QC                   := "Z025");
_002: NOP   0;
NETWORK
TITLE = Blocks AIN, GBA33, 026, 623, 624
      A(;
      A(;
      CALL  "AIN" , "AIN_VALs_VIB" (
           IN                       := "VB2_W",
           OUT                      := "VB2");
      A     BR;
      );
      JNB   _003;
      CALL  "GAINBI" (
           IN                       := "VB2",
           PARA_VAl                 := "GAINBI-VALs".Param_GBA35,
           OUT                      := "VBA2");
_003: A     BR;
      );
      JNB   _004;
      CALL  "2xHISIGMTV, QC" (
           INPUT                    := "VBA2",
           STPT_1                   := "VIBLIMIT",
           STPT_2                   := "VIBTRIP",
           Param_1                  := "HISIGMTV-VALs".Param_622,
           Param_2                  := "HISIGMTV-VALs".Param_623,
           OUT_1                    := "VBALM2",
           OUT_2                    := "VBTRP2",
           OUT_QC                   := "Z026");
_004: NOP   0;
NETWORK
TITLE = Blocks AIN, GBA34, 027, 625, 626
      A(;
      A(;
      CALL  "AIN" , "AIN_VALs_VIB" (
           IN                       := "VB3_W",
           OUT                      := "VB3");
      A     BR;
      );
      JNB   _005;
      CALL  "GAINBI" (
           IN                       := "VB3",
           PARA_VAl                 := "GAINBI-VALs".Param_GBA36,
           OUT                      := "VBA3");
_005: A     BR;
      );
      JNB   _006;
      CALL  "2xHISIGMTV, QC" (
           INPUT                    := "VBA3",
           STPT_1                   := "VIBLIMIT",
           STPT_2                   := "VIBTRIP",
           Param_1                  := "HISIGMTV-VALs".Param_624,
           Param_2                  := "HISIGMTV-VALs".Param_625,
           OUT_1                    := "VBALM3",
           OUT_2                    := "VBTRP3",
           OUT_QC                   := "Z027");
_006: NOP   0;
NETWORK
TITLE = Blocks AIN, GBA35, 028, 627, 628
      A(;
      A(;
      CALL  "AIN" , "AIN_VALs_VIB" (
           IN                       := "VB4_W",
           OUT                      := "VB4");
      A     BR;
      );
      JNB   _007;
      CALL  "GAINBI" (
           IN                       := "VB4",
           PARA_VAl                 := "GAINBI-VALs".Param_GBA37,
           OUT                      := "VBA4");
_007: A     BR;
      );
      JNB   _008;
      CALL  "2xHISIGMTV, QC" (
           INPUT                    := "VBA4",
           STPT_1                   := "VIBLIMIT",
           STPT_2                   := "VIBTRIP",
           Param_1                  := "HISIGMTV-VALs".Param_626,
           Param_2                  := "HISIGMTV-VALs".Param_627,
           OUT_1                    := "VBALM4",
           OUT_2                    := "VBTRP4",
           OUT_QC                   := "Z028");
_008: NOP   0;
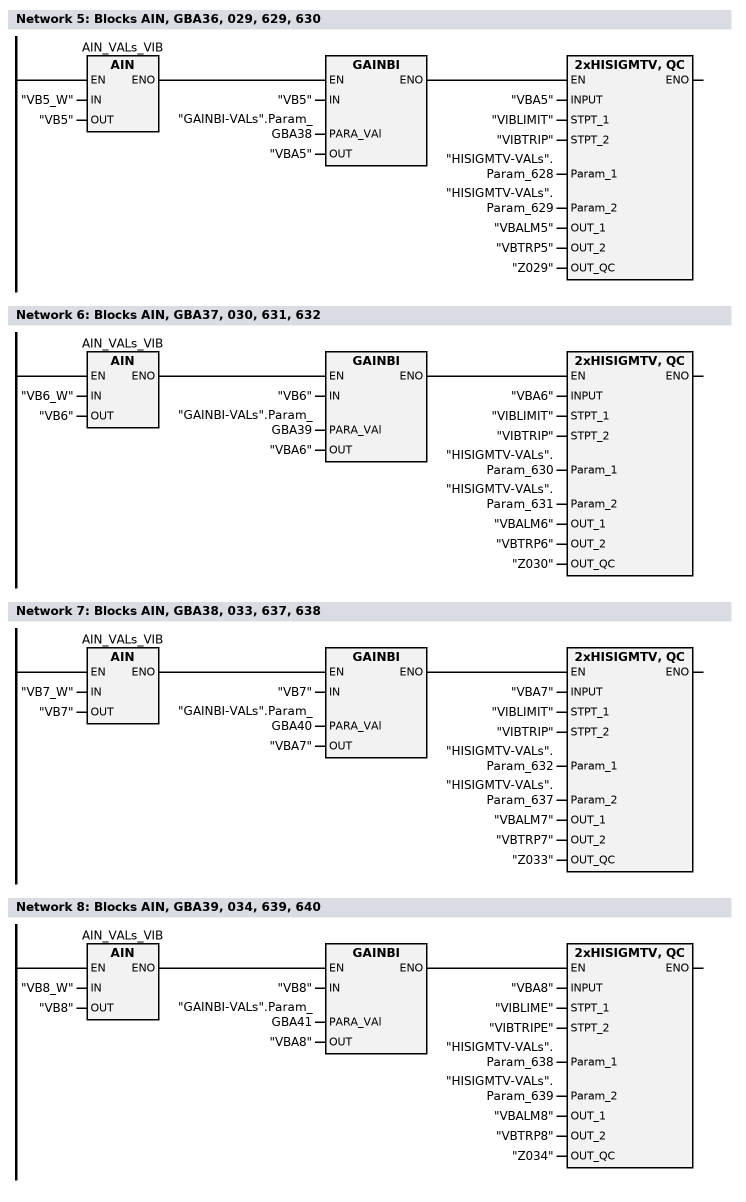
NETWORK
TITLE = Blocks AIN, GBA36, 029, 629, 630
      A(;
      A(;
      CALL  "AIN" , "AIN_VALs_VIB" (
           IN                       := "VB5_W",
           OUT                      := "VB5");
      A     BR;
      );
      JNB   _009;
      CALL  "GAINBI" (
           IN                       := "VB5",
           PARA_VAl                 := "GAINBI-VALs".Param_GBA38,
           OUT                      := "VBA5");
_009: A     BR;
      );
      JNB   _00a;
      CALL  "2xHISIGMTV, QC" (
           INPUT                    := "VBA5",
           STPT_1                   := "VIBLIMIT",
           STPT_2                   := "VIBTRIP",
           Param_1                  := "HISIGMTV-VALs".Param_628,
           Param_2                  := "HISIGMTV-VALs".Param_629,
           OUT_1                    := "VBALM5",
           OUT_2                    := "VBTRP5",
           OUT_QC                   := "Z029");
_00a: NOP   0;
NETWORK
TITLE = Blocks AIN, GBA37, 030, 631, 632
      A(;
      A(;
      CALL  "AIN" , "AIN_VALs_VIB" (
           IN                       := "VB6_W",
           OUT                      := "VB6");
      A     BR;
      );
      JNB   _00b;
      CALL  "GAINBI" (
           IN                       := "VB6",
           PARA_VAl                 := "GAINBI-VALs".Param_GBA39,
           OUT                      := "VBA6");
_00b: A     BR;
      );
      JNB   _00c;
      CALL  "2xHISIGMTV, QC" (
           INPUT                    := "VBA6",
           STPT_1                   := "VIBLIMIT",
           STPT_2                   := "VIBTRIP",
           Param_1                  := "HISIGMTV-VALs".Param_630,
           Param_2                  := "HISIGMTV-VALs".Param_631,
           OUT_1                    := "VBALM6",
           OUT_2                    := "VBTRP6",
           OUT_QC                   := "Z030");
_00c: NOP   0;
NETWORK
TITLE = Blocks AIN, GBA38, 033, 637, 638
      A(;
      A(;
      CALL  "AIN" , "AIN_VALs_VIB" (
           IN                       := "VB7_W",
           OUT                      := "VB7");
      A     BR;
      );
      JNB   _00d;
      CALL  "GAINBI" (
           IN                       := "VB7",
           PARA_VAl                 := "GAINBI-VALs".Param_GBA40,
           OUT                      := "VBA7");
_00d: A     BR;
      );
      JNB   _00e;
      CALL  "2xHISIGMTV, QC" (
           INPUT                    := "VBA7",
           STPT_1                   := "VIBLIMIT",
           STPT_2                   := "VIBTRIP",
           Param_1                  := "HISIGMTV-VALs".Param_632,
           Param_2                  := "HISIGMTV-VALs".Param_637,
           OUT_1                    := "VBALM7",
           OUT_2                    := "VBTRP7",
           OUT_QC                   := "Z033");
_00e: NOP   0;
NETWORK
TITLE = Blocks AIN, GBA39, 034, 639, 640
      A(;
      A(;
      CALL  "AIN" , "AIN_VALs_VIB" (
           IN                       := "VB8_W",
           OUT                      := "VB8");
      A     BR;
      );
      JNB   _00f;
      CALL  "GAINBI" (
           IN                       := "VB8",
           PARA_VAl                 := "GAINBI-VALs".Param_GBA41,
           OUT                      := "VBA8");
_00f: A     BR;
      );
      JNB   _010;
      CALL  "2xHISIGMTV, QC" (
           INPUT                    := "VBA8",
           STPT_1                   := "VIBLIME",
           STPT_2                   := "VIBTRIPE",
           Param_1                  := "HISIGMTV-VALs".Param_638,
           Param_2                  := "HISIGMTV-VALs".Param_639,
           OUT_1                    := "VBALM8",
           OUT_2                    := "VBTRP8",
           OUT_QC                   := "Z034");
_010: NOP   0;
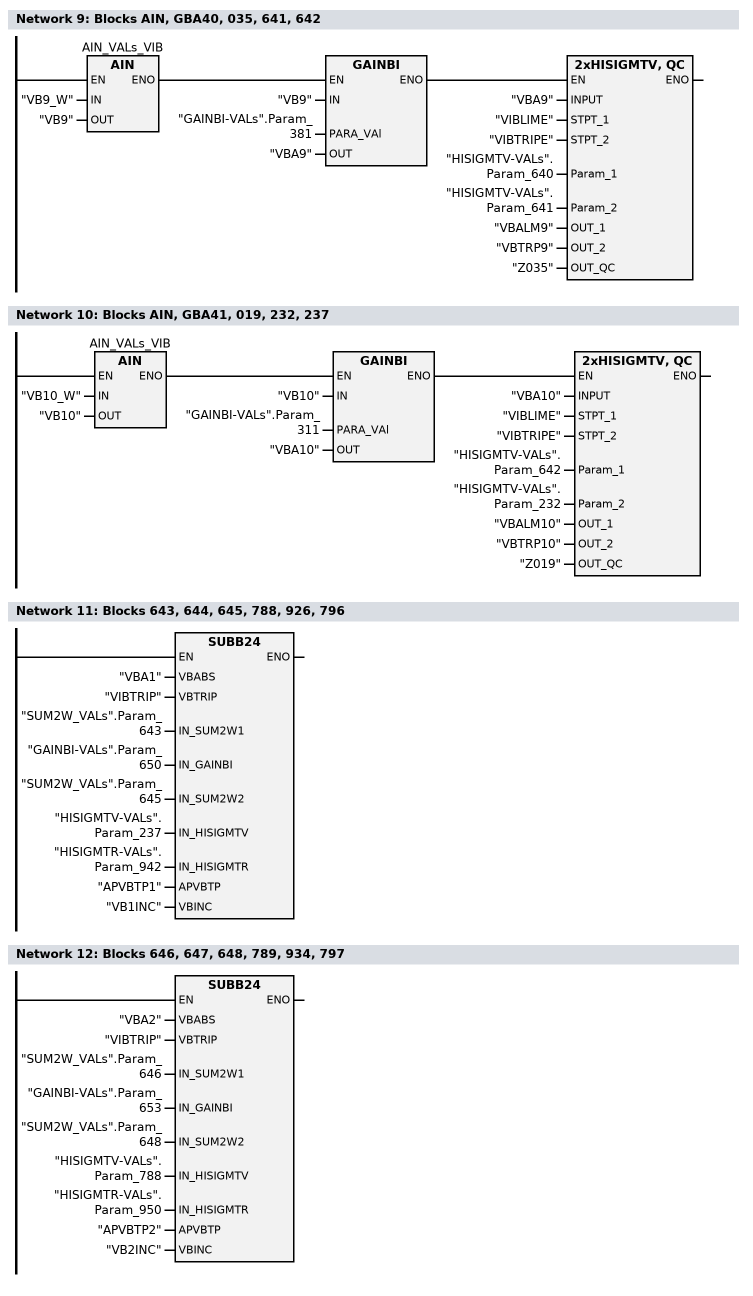
NETWORK
TITLE = Blocks AIN, GBA40, 035, 641, 642
      A(;
      A(;
      CALL  "AIN" , "AIN_VALs_VIB" (
           IN                       := "VB9_W",
           OUT                      := "VB9");
      A     BR;
      );
      JNB   _011;
      CALL  "GAINBI" (
           IN                       := "VB9",
           PARA_VAl                 := "GAINBI-VALs".Param_381,
           OUT                      := "VBA9");
_011: A     BR;
      );
      JNB   _012;
      CALL  "2xHISIGMTV, QC" (
           INPUT                    := "VBA9",
           STPT_1                   := "VIBLIME",
           STPT_2                   := "VIBTRIPE",
           Param_1                  := "HISIGMTV-VALs".Param_640,
           Param_2                  := "HISIGMTV-VALs".Param_641,
           OUT_1                    := "VBALM9",
           OUT_2                    := "VBTRP9",
           OUT_QC                   := "Z035");
_012: NOP   0;
NETWORK
TITLE = Blocks AIN, GBA41, 019, 232, 237
      A(;
      A(;
      CALL  "AIN" , "AIN_VALs_VIB" (
           IN                       := "VB10_W",
           OUT                      := "VB10");
      A     BR;
      );
      JNB   _013;
      CALL  "GAINBI" (
           IN                       := "VB10",
           PARA_VAl                 := "GAINBI-VALs".Param_311,
           OUT                      := "VBA10");
_013: A     BR;
      );
      JNB   _014;
      CALL  "2xHISIGMTV, QC" (
           INPUT                    := "VBA10",
           STPT_1                   := "VIBLIME",
           STPT_2                   := "VIBTRIPE",
           Param_1                  := "HISIGMTV-VALs".Param_642,
           Param_2                  := "HISIGMTV-VALs".Param_232,
           OUT_1                    := "VBALM10",
           OUT_2                    := "VBTRP10",
           OUT_QC                   := "Z019");
_014: NOP   0;
NETWORK
TITLE = Blocks 643, 644, 645, 788, 926, 796
      CALL  "SUBB24" (
           VBABS                    := "VBA1",
           VBTRIP                   := "VIBTRIP",
           IN_SUM2W1                := "SUM2W_VALs".Param_643,
           IN_GAINBI                := "GAINBI-VALs".Param_650,
           IN_SUM2W2                := "SUM2W_VALs".Param_645,
           IN_HISIGMTV              := "HISIGMTV-VALs".Param_237,
           IN_HISIGMTR              := "HISIGMTR-VALs".Param_942,
           APVBTP                   := "APVBTP1",
           VBINC                    := "VB1INC");
      NOP   0;
NETWORK
TITLE = Blocks 646, 647, 648, 789, 934, 797
      CALL  "SUBB24" (
           VBABS                    := "VBA2",
           VBTRIP                   := "VIBTRIP",
           IN_SUM2W1                := "SUM2W_VALs".Param_646,
           IN_GAINBI                := "GAINBI-VALs".Param_653,
           IN_SUM2W2                := "SUM2W_VALs".Param_648,
           IN_HISIGMTV              := "HISIGMTV-VALs".Param_788,
           IN_HISIGMTR              := "HISIGMTR-VALs".Param_950,
           APVBTP                   := "APVBTP2",
           VBINC                    := "VB2INC");
      NOP   0;
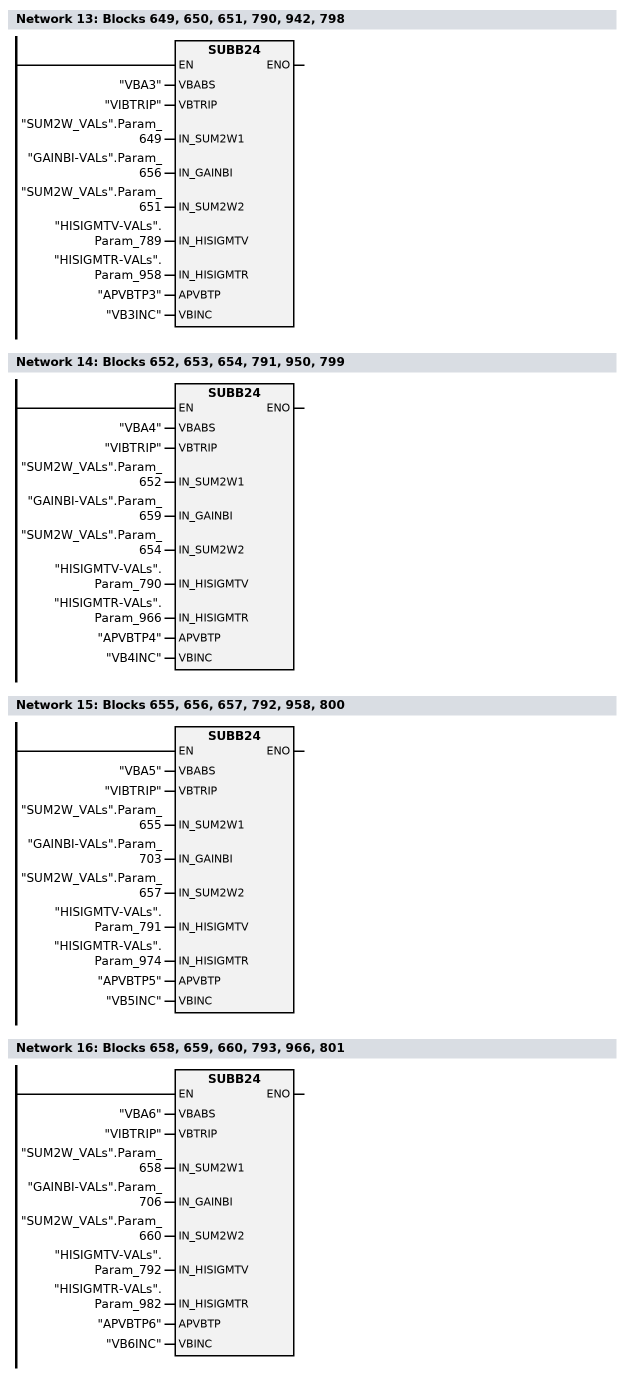
NETWORK
TITLE = Blocks 649, 650, 651, 790, 942, 798
      CALL  "SUBB24" (
           VBABS                    := "VBA3",
           VBTRIP                   := "VIBTRIP",
           IN_SUM2W1                := "SUM2W_VALs".Param_649,
           IN_GAINBI                := "GAINBI-VALs".Param_656,
           IN_SUM2W2                := "SUM2W_VALs".Param_651,
           IN_HISIGMTV              := "HISIGMTV-VALs".Param_789,
           IN_HISIGMTR              := "HISIGMTR-VALs".Param_958,
           APVBTP                   := "APVBTP3",
           VBINC                    := "VB3INC");
      NOP   0;
NETWORK
TITLE = Blocks 652, 653, 654, 791, 950, 799
      CALL  "SUBB24" (
           VBABS                    := "VBA4",
           VBTRIP                   := "VIBTRIP",
           IN_SUM2W1                := "SUM2W_VALs".Param_652,
           IN_GAINBI                := "GAINBI-VALs".Param_659,
           IN_SUM2W2                := "SUM2W_VALs".Param_654,
           IN_HISIGMTV              := "HISIGMTV-VALs".Param_790,
           IN_HISIGMTR              := "HISIGMTR-VALs".Param_966,
           APVBTP                   := "APVBTP4",
           VBINC                    := "VB4INC");
      NOP   0;
NETWORK
TITLE = Blocks 655, 656, 657, 792, 958, 800
      CALL  "SUBB24" (
           VBABS                    := "VBA5",
           VBTRIP                   := "VIBTRIP",
           IN_SUM2W1                := "SUM2W_VALs".Param_655,
           IN_GAINBI                := "GAINBI-VALs".Param_703,
           IN_SUM2W2                := "SUM2W_VALs".Param_657,
           IN_HISIGMTV              := "HISIGMTV-VALs".Param_791,
           IN_HISIGMTR              := "HISIGMTR-VALs".Param_974,
           APVBTP                   := "APVBTP5",
           VBINC                    := "VB5INC");
      NOP   0;
NETWORK
TITLE = Blocks 658, 659, 660, 793, 966, 801
      CALL  "SUBB24" (
           VBABS                    := "VBA6",
           VBTRIP                   := "VIBTRIP",
           IN_SUM2W1                := "SUM2W_VALs".Param_658,
           IN_GAINBI                := "GAINBI-VALs".Param_706,
           IN_SUM2W2                := "SUM2W_VALs".Param_660,
           IN_HISIGMTV              := "HISIGMTV-VALs".Param_792,
           IN_HISIGMTR              := "HISIGMTR-VALs".Param_982,
           APVBTP                   := "APVBTP6",
           VBINC                    := "VB6INC");
      NOP   0;
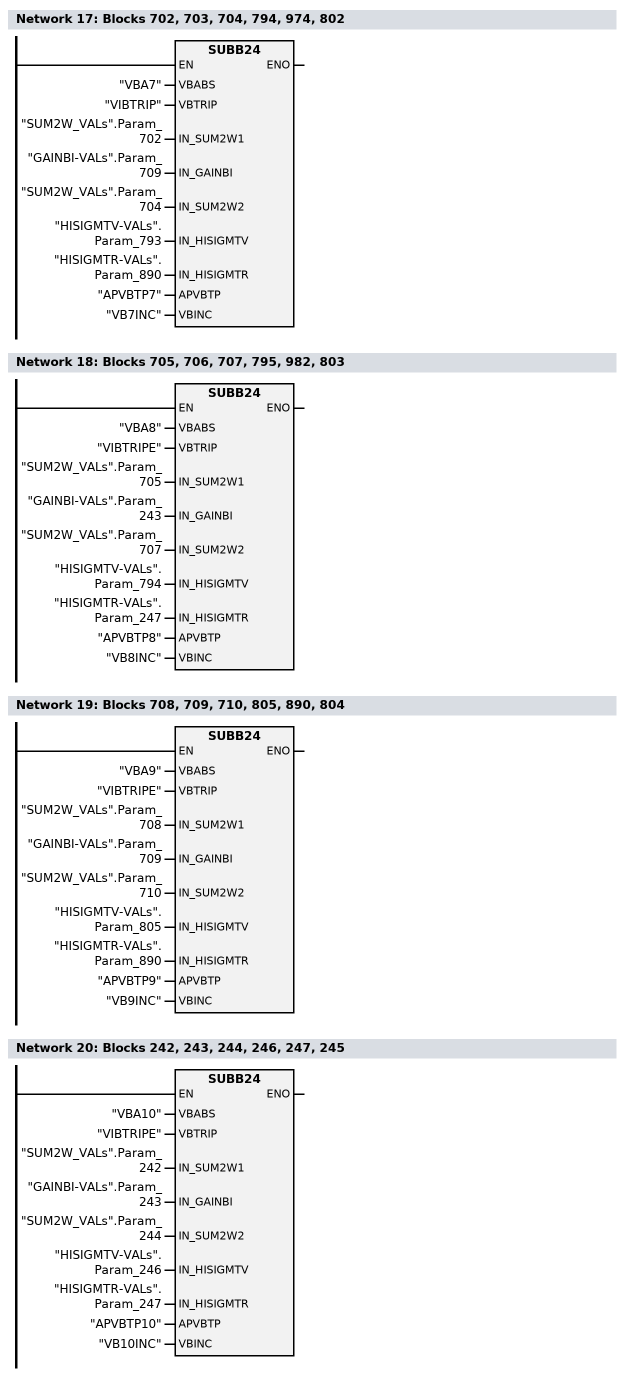
NETWORK
TITLE = Blocks 702, 703, 704, 794, 974, 802
      CALL  "SUBB24" (
           VBABS                    := "VBA7",
           VBTRIP                   := "VIBTRIP",
           IN_SUM2W1                := "SUM2W_VALs".Param_702,
           IN_GAINBI                := "GAINBI-VALs".Param_709,
           IN_SUM2W2                := "SUM2W_VALs".Param_704,
           IN_HISIGMTV              := "HISIGMTV-VALs".Param_793,
           IN_HISIGMTR              := "HISIGMTR-VALs".Param_890,
           APVBTP                   := "APVBTP7",
           VBINC                    := "VB7INC");
      NOP   0;
NETWORK
TITLE = Blocks 705, 706, 707, 795, 982, 803
      CALL  "SUBB24" (
           VBABS                    := "VBA8",
           VBTRIP                   := "VIBTRIPE",
           IN_SUM2W1                := "SUM2W_VALs".Param_705,
           IN_GAINBI                := "GAINBI-VALs".Param_243,
           IN_SUM2W2                := "SUM2W_VALs".Param_707,
           IN_HISIGMTV              := "HISIGMTV-VALs".Param_794,
           IN_HISIGMTR              := "HISIGMTR-VALs".Param_247,
           APVBTP                   := "APVBTP8",
           VBINC                    := "VB8INC");
      NOP   0;
NETWORK
TITLE = Blocks 708, 709, 710, 805, 890, 804
      CALL  "SUBB24" (
           VBABS                    := "VBA9",
           VBTRIP                   := "VIBTRIPE",
           IN_SUM2W1                := "SUM2W_VALs".Param_708,
           IN_GAINBI                := "GAINBI-VALs".Param_709,
           IN_SUM2W2                := "SUM2W_VALs".Param_710,
           IN_HISIGMTV              := "HISIGMTV-VALs".Param_805,
           IN_HISIGMTR              := "HISIGMTR-VALs".Param_890,
           APVBTP                   := "APVBTP9",
           VBINC                    := "VB9INC");
      NOP   0;
NETWORK
TITLE = Blocks 242, 243, 244, 246, 247, 245
      CALL  "SUBB24" (
           VBABS                    := "VBA10",
           VBTRIP                   := "VIBTRIPE",
           IN_SUM2W1                := "SUM2W_VALs".Param_242,
           IN_GAINBI                := "GAINBI-VALs".Param_243,
           IN_SUM2W2                := "SUM2W_VALs".Param_244,
           IN_HISIGMTV              := "HISIGMTV-VALs".Param_246,
           IN_HISIGMTR              := "HISIGMTR-VALs".Param_247,
           APVBTP                   := "APVBTP10",
           VBINC                    := "VB10INC");
      NOP   0;
END_FUNCTION

FUNCTION "TOD_Conversion" : VOID	// FC 3
VERSION : 0.0
VAR_INPUT
  CTime : TIME_OF_DAY ;
END_VAR
VAR_OUTPUT
  Hours : INT ;
  Minutes : INT ;
  Seconds : INT ;
END_VAR
VAR_TEMP
  INT_Time : DINT ;
  A : DINT ;
  B : DINT ;
END_VAR
BEGIN
// body was compiled from an SCL source; compiled code not shown
END_FUNCTION

FUNCTION "Sheet 2 (RSM)" : VOID	// FC 4
TITLE = Sheet 2 (RSM)
//Constants Initialization
AUTHOR : RJ
FAMILY : RSM
VERSION : 0.1
BEGIN
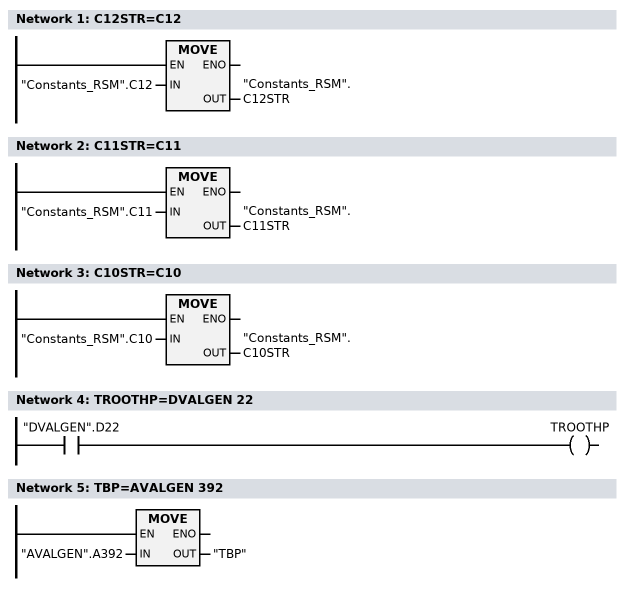
NETWORK
TITLE = C12STR=C12
      L     "Constants_RSM".C12;
      T     "Constants_RSM".C12STR;
      NOP   0;
NETWORK
TITLE = C11STR=C11
      L     "Constants_RSM".C11;
      T     "Constants_RSM".C11STR;
      NOP   0;
NETWORK
TITLE = C10STR=C10
      L     "Constants_RSM".C10;
      T     "Constants_RSM".C10STR;
      NOP   0;
NETWORK
TITLE = TROOTHP=DVALGEN 22
      A     "DVALGEN".D22;
      =     "TROOTHP";
NETWORK
TITLE = TBP=AVALGEN 392
      L     "AVALGEN".A392;
      T     "TBP";
      NOP   0;
END_FUNCTION

FUNCTION "TRANSF" : VOID	// FC 5
VERSION : 0.0
VAR_INPUT
  FLAG : BOOL ;
  IN1_y : REAL ;
  IN2_n : REAL ;
END_VAR
VAR_OUTPUT
  OUT : REAL ;
END_VAR
BEGIN
// body was compiled from an SCL source; compiled code not shown
END_FUNCTION

FUNCTION "AIFCTGEN" : VOID	// FC 6
AUTHOR : RJ
VERSION : 0.0
VAR_INPUT
  IN1 : REAL ;
  Parameters : STRUCT
   R : ARRAY  [1 .. 9 ] OF REAL ;
   S : ARRAY  [1 .. 9 ] OF REAL ;
   NMBP : INT ;
  END_STRUCT ;
END_VAR
VAR_OUTPUT
  OUT : REAL ;
END_VAR
VAR_TEMP
  i : INT ;
  Slope : REAL ;
  NMBP : INT ;
  R : ARRAY  [1 .. 9 ] OF REAL ;
  S : ARRAY  [1 .. 9 ] OF REAL ;
  Quality : BOOL ;	//1=Bad, 0=Fair
END_VAR
BEGIN
// body was compiled from an SCL source; compiled code not shown
END_FUNCTION

FUNCTION "BIN_SEARCH" : INT	// FC 7
AUTHOR : RJ
VERSION : 0.0
VAR_INPUT
  Size : INT ;
  A : ARRAY  [1 .. 9 ] OF REAL ;
  Key : REAL ;
END_VAR
VAR_OUTPUT
  RET_VAL : INT ;
END_VAR
VAR_TEMP
  bound : ARRAY  [1 .. 2 ] OF INT ;
  n : INT ;
END_VAR
BEGIN
// body was compiled from an SCL source; compiled code not shown
END_FUNCTION

FUNCTION "XHISEL" : VOID	// FC 8
VERSION : 0.0
VAR_INPUT
  PV : REAL ;
  CAS : REAL ;
  Param : STRUCT
   PV_GAIN : REAL ;
   PV_BIAS : REAL ;
   CAS_GAIN : REAL ;
   CAS_BIAS : REAL ;
   SCALE_TOP : REAL ;
   SCALE_BOT : REAL ;
  END_STRUCT ;
END_VAR
VAR_OUTPUT
  OUT : REAL ;
END_VAR
VAR_TEMP
  PVGB : REAL ;
  CASGB : REAL ;
  PV_GAIN : REAL ;
  PV_BIAS : REAL ;
  CAS_GAIN : REAL ;
  CAS_BIAS : REAL ;
  SCALE_TOP : REAL ;
  SCALE_BOT : REAL ;
END_VAR
BEGIN
// body was compiled from an SCL source; compiled code not shown
END_FUNCTION

FUNCTION "QAVGN" : VOID	// FC 10
VERSION : 0.0
VAR_INPUT
  IN1 : REAL ;
  IN2 : REAL ;
END_VAR
VAR_OUTPUT
  OUT : REAL ;
END_VAR
VAR_TEMP
  Temp : REAL ;
END_VAR
BEGIN
// body was compiled from an SCL source; compiled code not shown
END_FUNCTION

FUNCTION "HISIGMTR" : VOID	// FC 11
AUTHOR : Sabeeh
VERSION : 0.0
VAR_INPUT
  IN : REAL ;
  PARA_VAl : STRUCT
   STPT : REAL ;
   DBAN : REAL ;
  END_STRUCT ;
END_VAR
VAR_OUTPUT
  OUT : BOOL ;
END_VAR
BEGIN
// body was compiled from an SCL source; compiled code not shown
END_FUNCTION

FUNCTION "LOSIGMTR" : VOID	// FC 12
AUTHOR : Sabeeh
VERSION : 0.0
VAR_INPUT
  IN : REAL ;
  PARA_VAl : STRUCT
   STPT : REAL ;
   DBAN : REAL ;
  END_STRUCT ;
END_VAR
VAR_OUTPUT
  OUT : BOOL ;
END_VAR
BEGIN
// body was compiled from an SCL source; compiled code not shown
END_FUNCTION

FUNCTION "GAINBI" : VOID	// FC 14
AUTHOR : Sabeeh
VERSION : 0.0
VAR_INPUT
  IN : REAL ;
  PARA_VAl : STRUCT
   GAIN : REAL ;
   BIAS : REAL ;
  END_STRUCT ;
END_VAR
VAR_OUTPUT
  OUT : REAL ;
END_VAR
BEGIN
// body was compiled from an SCL source; compiled code not shown
END_FUNCTION

FUNCTION "DELTAW" : VOID	// FC 15
AUTHOR : Sabeeh
VERSION : 0.0
VAR_INPUT
  IN1_p : REAL ;
  IN2_n : REAL ;
  PARA_VAl : STRUCT
   WT1 : REAL ;
   WT2 : REAL ;
  END_STRUCT ;
END_VAR
VAR_OUTPUT
  OUT : REAL ;
END_VAR
BEGIN
// body was compiled from an SCL source; compiled code not shown
END_FUNCTION

FUNCTION "HILOLMTV" : VOID	// FC 16
AUTHOR : Sabeeh
VERSION : 0.0
VAR_INPUT
  IN : REAL ;
  PARA_VAl : STRUCT
   LOLM : REAL ;
   HILM : REAL ;
  END_STRUCT ;
END_VAR
VAR_OUTPUT
  OUT : REAL ;
END_VAR
BEGIN
// body was compiled from an SCL source; compiled code not shown
END_FUNCTION

FUNCTION "HILOMTR" : VOID	// FC 18
AUTHOR : Sabeeh
VERSION : 0.0
VAR_INPUT
  IN : REAL ;
  PARA_VAl : STRUCT
   HISP : REAL ;
   HIDB : REAL ;
   LOSP : REAL ;
   LODB : REAL ;
  END_STRUCT ;
END_VAR
VAR_OUTPUT
  OUT : BOOL ;
END_VAR
BEGIN
// body was compiled from an SCL source; compiled code not shown
END_FUNCTION

FUNCTION "QTRANSN" : VOID	// FC 19
VERSION : 0.0
VAR_INPUT
  IN1 : REAL ;
  IN2 : REAL ;
END_VAR
VAR_OUTPUT
  OUT : REAL ;
END_VAR
BEGIN
// body was compiled from an SCL source; compiled code not shown
END_FUNCTION

FUNCTION "DIVIDEGB" : VOID	// FC 21
AUTHOR : RJ
VERSION : 0.0
VAR_INPUT
  IN1_Top : REAL ;
  IN2_Side : REAL ;
  Param : STRUCT
   GAIN : REAL ;
   BIAS : REAL ;
  END_STRUCT ;
END_VAR
VAR_OUTPUT
  OUT : REAL ;
END_VAR
VAR_TEMP
  GAIN : REAL ;
  BIAS : REAL ;
END_VAR
BEGIN
// body was compiled from an SCL source; compiled code not shown
END_FUNCTION

FUNCTION "POLY" : VOID	// FC 22
AUTHOR : RJ
VERSION : 0.0
VAR_INPUT
  IN : REAL ;
  Param : STRUCT
   CX0 : REAL ;
   CX1 : REAL ;
   CX2 : REAL ;
   CX3 : REAL ;
   CX4 : REAL ;
   CX5 : REAL ;
  END_STRUCT ;
END_VAR
VAR_OUTPUT
  OUT : REAL ;
END_VAR
VAR_TEMP
  CX0 : REAL ;
  CX1 : REAL ;
  CX2 : REAL ;
  CX3 : REAL ;
  CX4 : REAL ;
  CX5 : REAL ;
END_VAR
BEGIN
// body was compiled from an SCL source; compiled code not shown
END_FUNCTION

FUNCTION "QBLOCK" : VOID	// FC 23
AUTHOR : RJ
VERSION : 0.0
VAR_INPUT
  IN : REAL ;
END_VAR
VAR_OUTPUT
  OUT : REAL ;
END_VAR
BEGIN
// body was compiled from an SCL source; compiled code not shown
END_FUNCTION

FUNCTION "SUM8W" : VOID	// FC 24
AUTHOR : RJ
VERSION : 0.0
VAR_INPUT
  IN1 : REAL ;
  IN2 : REAL ;
  IN3 : REAL ;
  IN4 : REAL ;
  IN5 : REAL ;
  IN6 : REAL ;
  IN7 : REAL ;
  IN8 : REAL ;
  Param : STRUCT
   WT1 : REAL ;
   WT2 : REAL ;
   WT3 : REAL ;
   WT4 : REAL ;
   WT5 : REAL ;
   WT6 : REAL ;
   WT7 : REAL ;
   WT8 : REAL ;
  END_STRUCT ;
END_VAR
VAR_OUTPUT
  OUT : REAL ;
END_VAR
VAR_TEMP
  WT1 : REAL ;
  WT2 : REAL ;
  WT3 : REAL ;
  WT4 : REAL ;
  WT5 : REAL ;
  WT6 : REAL ;
  WT7 : REAL ;
  WT8 : REAL ;
END_VAR
BEGIN
// body was compiled from an SCL source; compiled code not shown
END_FUNCTION

FUNCTION "Sheet 3 (RSM)" : VOID	// FC 25
TITLE = Sheet 3 (RSM)
//FSST & TIMP & TSAT (Analog)
AUTHOR : RJ
FAMILY : RSM
VERSION : 0.1
BEGIN
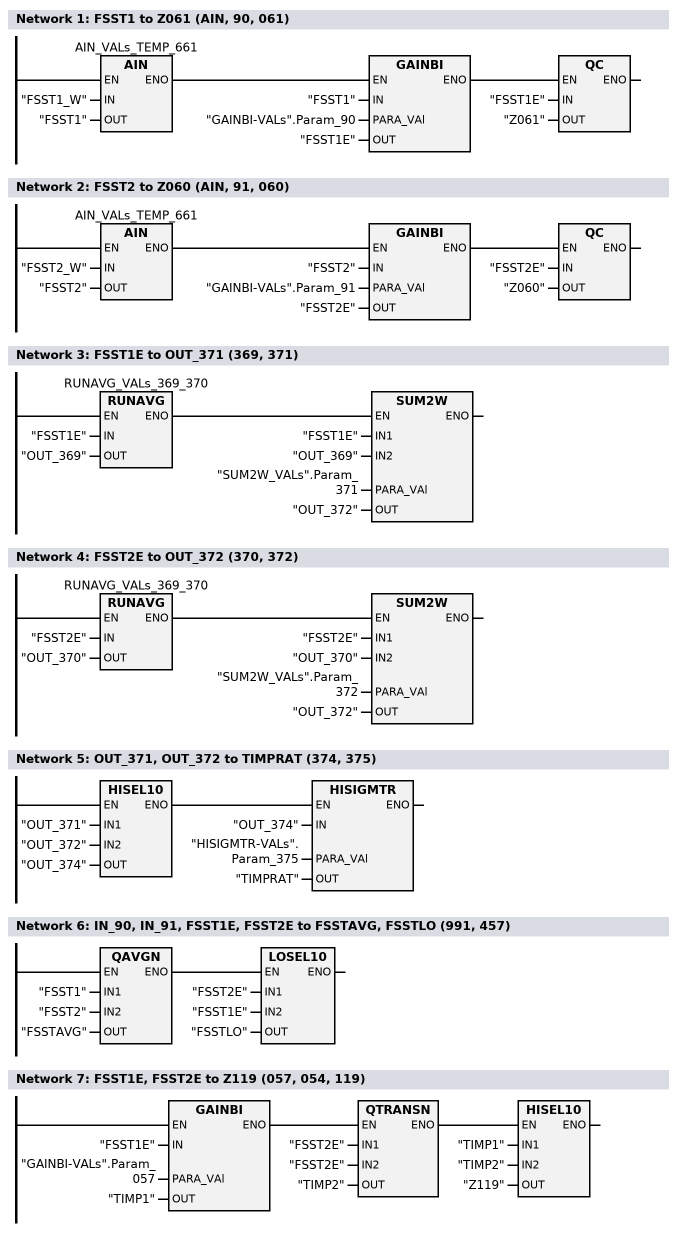
NETWORK
TITLE = FSST1 to Z061 (AIN, 90, 061)
      A(;
      A(;
      CALL  "AIN" , "AIN_VALs_TEMP_661" (
           IN                       := "FSST1_W",
           OUT                      := "FSST1");
      A     BR;
      );
      JNB   _001;
      CALL  "GAINBI" (
           IN                       := "FSST1",
           PARA_VAl                 := "GAINBI-VALs".Param_90,
           OUT                      := "FSST1E");
_001: A     BR;
      );
      JNB   _002;
      CALL  "QC" (
           IN                       := "FSST1E",
           OUT                      := "Z061");
_002: NOP   0;
NETWORK
TITLE = FSST2 to Z060 (AIN, 91, 060)
      A(;
      A(;
      CALL  "AIN" , "AIN_VALs_TEMP_661" (
           IN                       := "FSST2_W",
           OUT                      := "FSST2");
      A     BR;
      );
      JNB   _003;
      CALL  "GAINBI" (
           IN                       := "FSST2",
           PARA_VAl                 := "GAINBI-VALs".Param_91,
           OUT                      := "FSST2E");
_003: A     BR;
      );
      JNB   _004;
      CALL  "QC" (
           IN                       := "FSST2E",
           OUT                      := "Z060");
_004: NOP   0;
NETWORK
TITLE = FSST1E to OUT_371 (369, 371)
      A(;
      CALL  "RUNAVG" , "RUNAVG_VALs_369_370" (
           IN                       := "FSST1E",
           OUT                      := "OUT_369");
      A     BR;
      );
      JNB   _005;
      CALL  "SUM2W" (
           IN1                      := "FSST1E",
           IN2                      := "OUT_369",
           PARA_VAl                 := "SUM2W_VALs".Param_371,
           OUT                      := "OUT_372");
_005: NOP   0;
NETWORK
TITLE = FSST2E to OUT_372 (370, 372)
      A(;
      CALL  "RUNAVG" , "RUNAVG_VALs_369_370" (
           IN                       := "FSST2E",
           OUT                      := "OUT_370");
      A     BR;
      );
      JNB   _006;
      CALL  "SUM2W" (
           IN1                      := "FSST2E",
           IN2                      := "OUT_370",
           PARA_VAl                 := "SUM2W_VALs".Param_372,
           OUT                      := "OUT_372");
_006: NOP   0;
NETWORK
TITLE = OUT_371, OUT_372 to TIMPRAT (374, 375)
      A(;
      CALL  "HISEL10" (
           IN1                      := "OUT_371",
           IN2                      := "OUT_372",
           OUT                      := "OUT_374");
      A     BR;
      );
      JNB   _007;
      CALL  "HISIGMTR" (
           IN                       := "OUT_374",
           PARA_VAl                 := "HISIGMTR-VALs".Param_375,
           OUT                      := "TIMPRAT");
_007: NOP   0;
NETWORK
TITLE = IN_90, IN_91, FSST1E, FSST2E to FSSTAVG, FSSTLO (991, 457) 
      A(;
      CALL  "QAVGN" (
           IN1                      := "FSST1",
           IN2                      := "FSST2",
           OUT                      := "FSSTAVG");
      A     BR;
      );
      JNB   _008;
      CALL  "LOSEL10" (
           IN1                      := "FSST2E",
           IN2                      := "FSST1E",
           OUT                      := "FSSTLO");
_008: NOP   0;
NETWORK
TITLE = FSST1E, FSST2E to Z119 (057, 054, 119)
      A(;
      A(;
      CALL  "GAINBI" (
           IN                       := "FSST1E",
           PARA_VAl                 := "GAINBI-VALs".Param_057,
           OUT                      := "TIMP1");
      A     BR;
      );
      JNB   _009;
      CALL  "QTRANSN" (
           IN1                      := "FSST2E",
           IN2                      := "FSST2E",
           OUT                      := "TIMP2");
_009: A     BR;
      );
      JNB   _00a;
      CALL  "HISEL10" (
           IN1                      := "TIMP1",
           IN2                      := "TIMP2",
           OUT                      := "Z119");
_00a: NOP   0;
NETWORK
TITLE = TMAX, Z119, Z115, TSAT, SELCO6 to TIMP (116, 120)
      A     "SELC06";
      =     L 0.0;
      BLD   103;
      A(;
      A     "Z115";
      =     L 0.1;
      BLD   103;
      CALL  "TRANSF" (
           FLAG                     := L 0.1,
           IN1_y                    := "TMAX",
           IN2_n                    := "Z119",
           OUT                      := "OUT_116");
      A     BR;
      );
      JNB   _00b;
      CALL  "TRANSF" (
           FLAG                     := L 0.0,
           IN1_y                    := "TSAT",
           IN2_n                    := "OUT_116",
           OUT                      := "TIMP");
_00b: NOP   0;
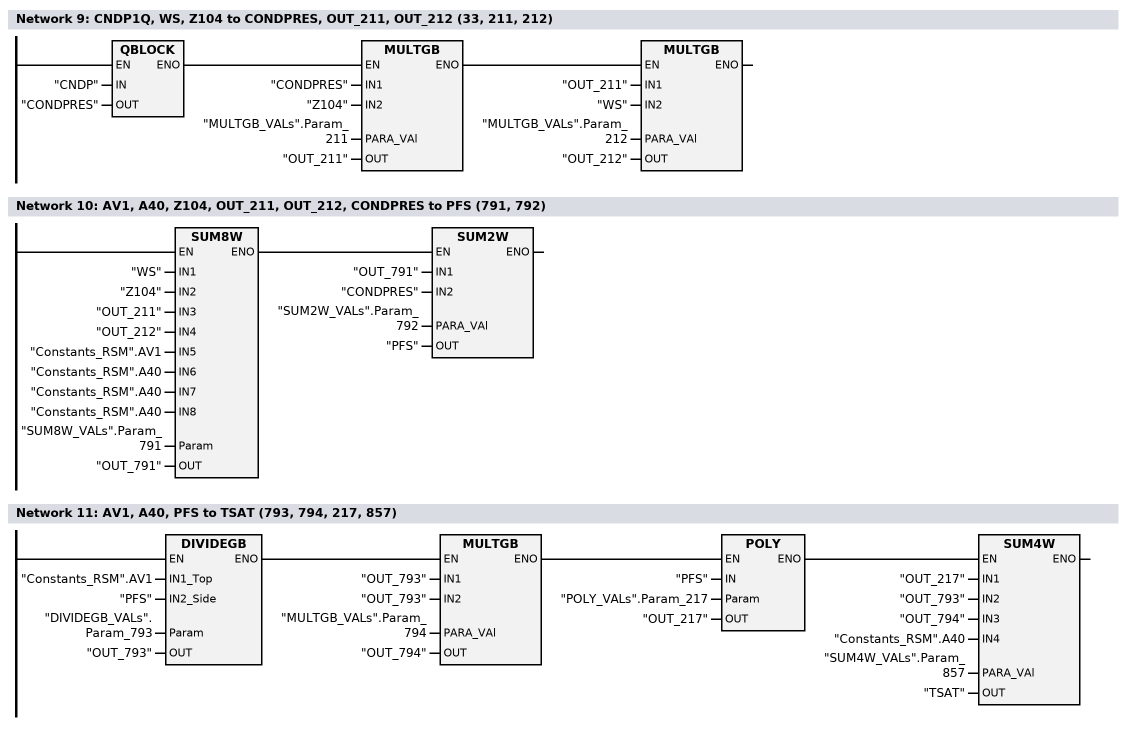
NETWORK
TITLE = CNDP1Q, WS, Z104 to CONDPRES, OUT_211, OUT_212 (33, 211, 212)
      A(;
      A(;
      CALL  "QBLOCK" (
           IN                       := "CNDP",
           OUT                      := "CONDPRES");
      A     BR;
      );
      JNB   _00c;
      CALL  "MULTGB" (
           IN1                      := "CONDPRES",
           IN2                      := "Z104",
           PARA_VAl                 := "MULTGB_VALs".Param_211,
           OUT                      := "OUT_211");
_00c: A     BR;
      );
      JNB   _00d;
      CALL  "MULTGB" (
           IN1                      := "OUT_211",
           IN2                      := "WS",
           PARA_VAl                 := "MULTGB_VALs".Param_212,
           OUT                      := "OUT_212");
_00d: NOP   0;
NETWORK
TITLE = AV1, A40, Z104, OUT_211, OUT_212, CONDPRES to PFS (791, 792)
      A(;
      CALL  "SUM8W" (
           IN1                      := "WS",
           IN2                      := "Z104",
           IN3                      := "OUT_211",
           IN4                      := "OUT_212",
           IN5                      := "Constants_RSM".AV1,
           IN6                      := "Constants_RSM".A40,
           IN7                      := "Constants_RSM".A40,
           IN8                      := "Constants_RSM".A40,
           Param                    := "SUM8W_VALs".Param_791,
           OUT                      := "OUT_791");
      A     BR;
      );
      JNB   _00e;
      CALL  "SUM2W" (
           IN1                      := "OUT_791",
           IN2                      := "CONDPRES",
           PARA_VAl                 := "SUM2W_VALs".Param_792,
           OUT                      := "PFS");
_00e: NOP   0;
NETWORK
TITLE = AV1, A40, PFS to TSAT (793, 794, 217, 857)
      A(;
      A(;
      A(;
      CALL  "DIVIDEGB" (
           IN1_Top                  := "Constants_RSM".AV1,
           IN2_Side                 := "PFS",
           Param                    := "DIVIDEGB_VALs".Param_793,
           OUT                      := "OUT_793");
      A     BR;
      );
      JNB   _00f;
      CALL  "MULTGB" (
           IN1                      := "OUT_793",
           IN2                      := "OUT_793",
           PARA_VAl                 := "MULTGB_VALs".Param_794,
           OUT                      := "OUT_794");
_00f: A     BR;
      );
      JNB   _010;
      CALL  "POLY" (
           IN                       := "PFS",
           Param                    := "POLY_VALs".Param_217,
           OUT                      := "OUT_217");
_010: A     BR;
      );
      JNB   _011;
      CALL  "SUM4W" (
           IN1                      := "OUT_217",
           IN2                      := "OUT_793",
           IN3                      := "OUT_794",
           IN4                      := "Constants_RSM".A40,
           PARA_VAl                 := "SUM4W_VALs".Param_857,
           OUT                      := "TSAT");
_011: NOP   0;
END_FUNCTION

